							iAutoAuxStep3:=888;
							iNGSize:=iNGSize+1;		
						END_IF	
				END_IF
			END_IF
	ELSE
		BeltData[BeltNo.OverHang].iPanoramaNG:=0;
		BeltData[BeltNo.OverHang].fPoleNGSizeNo:=CCD_COM.Size.fPoleNGSizeNo; 
		stAlarm.arrLightWarn[5]:=TRUE;//尺寸CCD检测超时，请查看！
		iAutoAuxStep3:=888;
		iNGSize:=iNGSize+1;
	END_IF
888://
;
END_CASE


///////////////////////////////////////////////////////////冲R角定位检测//////////////////////////////////////////////////////////////////
CASE iAutoAuxStep4 OF
10://
	IF arrAxisCtrl[VirAxisNo.VirMain].Status.fActPos < fRecordMouldCCDInMainPos-fRecordMouldCCDInMainPosMod+360+ProductPar.parPublic.fMainPos-10 THEN//到下个周期250度以前有效			
		IF arrAxisCtrl[VirAxisNo.VirMain].Status.fActPos>=fRecordMouldCCDInMainPos+30 THEN		
			IF CCD_COM.Chamfer.iFinish=1 THEN
				CutMark_R[0]:=FALSE;
				TabData[TabNo.MouldPhoto].fTab_OffsetM:=CCD_COM.Chamfer.fTabXOffset;
				TabData[TabNo.MouldPhoto].fTab_OffsetY:=CCD_COM.Chamfer.fTabYOffset; //20240524SJ
				iAutoAuxStep4:=888;
			ELSIF CCD_COM.Chamfer.iFinish=2 THEN
				CutMark_R[0]:=FALSE;
				TabData[TabNo.MouldPhoto].fTab_OffsetM:=CCD_COM.Chamfer.fTabXOffset;//CCD抓不到极耳时，给NG，纠偏量给1个片宽
				TabData[TabNo.MouldPhoto].fTab_OffsetY:=CCD_COM.Chamfer.fTabYOffset; //20240524SJ
				TabData[TabNo.MouldPhoto].bTabOffsetNG_M:=TRUE;
				//stAlarm.arrLightWarn[1]:=TRUE;//冲R角CCD定位检测NG，请查看！
				iAutoAuxStep4:=888;	
			ELSIF CCD_COM.Chamfer.iFinish=3 THEN
				TabData[TabNo.MouldPhoto].bTabOffsetNG_M:=TRUE;
				CutMark_R[0]:=TRUE;
				iAutoAuxStep4:=888;	
			END_IF	
		END_IF		
	ELSE			
		//TabData[TabNo.MouldPhoto].fTab_OffsetM:=PolePar.fPoleWidth;
		TabData[TabNo.MouldPhoto].fTab_OffsetM:=0;//20240524SJ
		TabData[TabNo.MouldPhoto].bTabOffsetNG_M:=TRUE;
		stAlarm.arrLightWarn[2]:=TRUE;//冲R角CCD定位检测超时，请查看！		
		iAutoAuxStep4:=889;			
	END_IF
888:
	;
END_CASE

///////////////////////////////////////////////////////////裁切定位检测////////////////////////////////////////////////////////////////////
CASE iAutoAuxStep5 OF
10://
	IF arrAxisCtrl[VirAxisNo.VirMain].Status.fActPos < fRecordCuterCCDInMainPos-fRecordCuterCCDInMainPosMod+360+ProductPar.parPublic.fMainPos-10 THEN//到下个周期250度以前有效			
		IF arrAxisCtrl[VirAxisNo.VirMain].Status.fActPos>=fRecordCuterCCDInMainPos+30 THEN		
			IF CCD_COM.Cuter.iFinish=1 THEN	
				TabData[TabNo.CuterPhoto].fTab_OffsetC:=CCD_COM.Cuter.fTabXOffset;
				InteData[InteNo.Cuter-2].fTabIntervalC:=CCD_COM.Cuter.fTabWidth;
				iAutoAuxStep5:=100;
			ELSIF CCD_COM.Cuter.iFinish=2 THEN	
				TabData[TabNo.CuterPhoto].fTab_OffsetC:=CCD_COM.Cuter.fTabXOffset;
				InteData[InteNo.Cuter-2].fTabIntervalC:=CCD_COM.Cuter.fTabWidth;//CCD抓不到极耳时，给NG，左侧相机纠偏量给1个片宽,,片宽给0
				InteData[InteNo.Cuter-2].bIntervalFail_C:=TRUE;
				TabData[TabNo.CuterPhoto].bTabOffsetNG_C:=TRUE;
				//stAlarm.arrLightWarn[3]:=TRUE;//裁切CCD定位检测NG，请查看！		
				iAutoAuxStep5:=888;
			ELSIF CCD_COM.Cuter.iFinish=3 THEN	
	                 	TabData[TabNo.CuterPhoto].fTab_OffsetC:=CCD_COM.Cuter.fTabXOffset;
				InteData[InteNo.Cuter-2].fTabIntervalC:=CCD_COM.Cuter.fTabWidth;//CCD抓不到极耳时，给NG，左侧相机纠偏量给1个片宽,,片宽给0
				InteData[InteNo.Cuter-2].bIntervalFail_C:=TRUE;
				TabData[TabNo.CuterPhoto].bTabOffsetNG_C:=TRUE;
				//stAlarm.arrLightWarn[3]:=TRUE;//裁切CCD定位检测NG，请查看！		
				iAutoAuxStep5:=888;					
			END_IF	
		END_IF		
	ELSE			
		TabData[TabNo.CuterPhoto].fTab_OffsetC:=PolePar.fPoleWidth;
		InteData[InteNo.Cuter-2].fTabIntervalC:=0;	
		InteData[InteNo.Cuter-2].bIntervalFail_C:=TRUE;
		TabData[TabNo.CuterPhoto].bTabOffsetNG_C:=TRUE;
		PolePar.AddAlarm  :=PolePar.AddAlarm +1;
		stAlarm.arrLightWarn[4]:=TRUE;//裁切CCD定位检测超时，请查看！					
		iAutoAuxStep5:=889;		
	END_IF
	
100:

	IF CCD_COM.Cuter.iFinish=1 AND ( ABS(CCD_COM.Cuter.fTabWidth-PolePar.TabWidthBace)>=0.5 ) THEN
		Production.NGFlag[15]:=TRUE;
		iTabWidth_JS:=iTabWidth_JS+1;
		iAutoAuxStep5:=200;	
	ELSE
		iTabWidth_JS:=0;
		iAutoAuxStep5:=300;	
	END_IF
200:		
	IF iTabWidth_JS >=10 AND NOT ProductPar.iModeEN.bTabWidtNGoff THEN
		stAlarm.arrFlowAlarm[41]:=TRUE;//极片来料不良，请检查
		iTabWidth_JS:=0;
	END_IF
	Production.NGFlag[15]:=FALSE;
	iAutoAuxStep5:=888;	

300:
	iTabWidth_JS:=0;
	iAutoAuxStep5:=888;	
888:
	;	
	
	
END_CASE

////////////////////////////////////////////////////////////////线扫拍照触发////////////////////////////////////////////////////////////////
ttLinePhoto(CLK:=arrAxisCtrl[VirAxisNo.VirMain].Status.fModuloSetPos>=2  
						AND arrAxisCtrl[VirAxisNo.VirMain].Status.fModuloSetPos<=6 
						AND  arrAxisCtrl[VirAxisNo.VirMain].Status.Moving 
						AND  stDriverCam.bInSync         , Q=> );
IF ttLinePhoto.Q THEN
	CCD_COM.Scan.bSendMark:=FALSE;//PLC_To_PC上位机的发送数据标志
	IF NOT ProductPar.iModeEN.bCcdTcpEN AND NOT ProductPar.iModeEN.bLineScanCCDEN  THEN//线扫OK信号
		
		CCD_COM.Scan.iResult_IO_UP:=33;//复位线扫IO结果
		CCD_COM.Scan.iResult_IO_Down:=33;
		bLineScanResult1_UP:=FALSE;
		bLineScanResult2_UP:=FALSE;
		bLineScanResult1_Down:=FALSE;
		bLineScanResult2_Down:=FALSE;
		CCD_IO.boXSPhoto:=TRUE;//自动线扫启动
		CCD_Com.iLineScanPhotoCount:=CCD_Com.iLineScanPhotoCount+1;
		IF  NOT  ProductPar.iLineScanSel THEN
	    	iAutoAuxStep11:=10;
		END_IF
		fRecordLineineScanCCDInMainPos:=arrAxisCtrl[VirAxisNo.VirMain].Status.fActPos;																								
		fRecordLineineScanCCDInMainPosMod:=arrAxisCtrl[VirAxisNo.VirMain].Status.fModuloActPos;		
	END_IF	
END_IF	

rLineScan_UPTCP(CLK:=CCD_COM.Scan.iResult_UP<>33      , Q=> );
rLineScan_DownTCP(CLK:=CCD_COM.Scan.iResult_Down<>33 , Q=> );

IF ProductPar.iLineScanSel THEN
     IF rLineScan_UPTCP.Q THEN
		 IF CCD_COM.Scan.iResult_UP<>0 THEN
		    CCD_Com.iLineScanReceiveResultCount_UP:=CCD_Com.iLineScanReceiveResultCount_UP+1;
		 END_IF
	 END_IF

     IF rLineScan_DownTCP.Q THEN
		  IF CCD_COM.Scan.iResult_Down<>0 THEN
		     CCD_Com.iLineScanReceiveResultCount_Down:=CCD_Com.iLineScanReceiveResultCount_Down+1;
		  END_IF
	 END_IF

ELSE 
			IF  rLineScanOK_UP.Q  OR rLineScanNG_UP.Q THEN
				CCD_Com.iLineScanReceiveResultCount_UP:=CCD_Com.iLineScanReceiveResultCount_UP+1;
				fDA1:=        arrAxisCtrl[VirAxisNo.VirMain].Status.fModuloActPos;
			END_IF

		    IF  rLineScanOK_Down.Q  OR rLineScanNG_Down.Q THEN
				CCD_Com.iLineScanReceiveResultCount_Down:=CCD_Com.iLineScanReceiveResultCount_Down+1;
				fDA2:=        arrAxisCtrl[VirAxisNo.VirMain].Status.fModuloActPos;
			END_IF

END_IF			
			
	IF CCD_Com.bLineScanPhotoCountClear THEN
       CCD_Com.iLineScanPhotoCount:=0;
	   CCD_Com.iLineScanReceiveResultCount_UP:=0;
	   CCD_Com.iLineScanReceiveResultCount_Down:=0;
    END_IF		
			
				
CASE iAutoAuxStep11 OF
10://
	IF arrAxisCtrl[VirAxisNo.VirMain].Status.fModuloActPos>5 AND arrAxisCtrl[VirAxisNo.VirMain].Status.fModuloActPos < ProductPar.parPublic.fMainPos-15 THEN//到下个周期判断结果前有效
			IF rLineScanOK_UP.Q THEN
				bLineScanResult1_UP:=TRUE;
			END_IF
			IF rLineScanNG_UP.Q THEN
				bLineScanResult2_UP:=TRUE;
			END_IF

			IF rLineScanOK_Down.Q THEN
				bLineScanResult1_Down:=TRUE;
			END_IF
			IF rLineScanNG_Down.Q THEN
				bLineScanResult2_Down:=TRUE;
			END_IF	
	
		IF (bLineScanResult1_UP OR bLineScanResult2_UP) AND (bLineScanResult1_Down OR bLineScanResult2_Down) THEN
			iAutoAuxStep11:=888;
		END_IF
	
	ELSIF  arrAxisCtrl[VirAxisNo.VirMain].Status.fModuloActPos > 320 THEN
		IF NOT (bLineScanResult1_UP OR bLineScanResult2_UP) AND (bLineScanResult1_Down OR bLineScanResult2_Down) THEN  //AND NOT ProductPar.iModeEN.bCcdTcpEN AND NOT ProductPar.iModeEN.bLineScanCCDEN
			stAlarm.arrFlowAlarm[25]:=TRUE;//上线扫超时报警
		END_IF
		IF (bLineScanResult1_UP OR bLineScanResult2_UP) AND NOT (bLineScanResult1_Down OR bLineScanResult2_Down) THEN//	AND NOT ProductPar.iModeEN.bCcdTcpEN AND NOT ProductPar.iModeEN.bLineScanCCDEN 
			stAlarm.arrFlowAlarm[27]:=TRUE;//下线扫超时报警
		END_IF
		iAutoAuxStep11:=886;
	END_IF
	
END_CASE

///////////////////////////////////////////////////////////CCD标定流程////////////////////////////////////////////////////////////////////
IF stSysState.iMode=3 THEN
	CASE iAutoAuxStep10 OF 
	0://
		IF 	CCD_IO.bCalibrationsDo THEN
			bChaNoPhoto:=FALSE;
			bCutNoPhoto:=FALSE;			
			iAutoAuxStep10:=10;
		ELSIF NOT CCD_IO.bCalibrationsDo AND CCD_IO.bCalibrationsDo_Cha AND NOT CCD_IO.bCalibrationsDo_Cut THEN
			bChaNoPhoto:=FALSE;
			bCutNoPhoto:=TRUE;
			iAutoAuxStep10:=10;
		ELSIF NOT CCD_IO.bCalibrationsDo AND NOT CCD_IO.bCalibrationsDo_Cha AND CCD_IO.bCalibrationsDo_Cut THEN
			bChaNoPhoto:=TRUE;
			bCutNoPhoto:=FALSE;			
			iAutoAuxStep10:=10;
		END_IF
	10://
		CCD_IO.bDemRuning:=TRUE;
		CCD_COM.iDemCount:=1;//是否需要延时
		iAutoAuxStep10:=20;
	20://
		IF NOT bChaNoPhoto THEN
			CCD_COM.iDemResult_Cha:=0;
			CCD_IO.hmiChamferPhoto:=TRUE;
		END_IF
		IF NOT bCutNoPhoto THEN
			CCD_COM.iDemResult_Cut:=0;
			CCD_IO.hmiCuterPhoto:=TRUE;
		END_IF	
		iAutoAuxStep10:=30;
	30://
		IF tonAuto[17].Q THEN
			CCD_IO.hmiChamferPhoto:=FALSE;
			CCD_IO.hmiCuterPhoto:=FALSE;
			tonAuto[18].IN:=FALSE;
			iAutoAuxStep10:=40;
		END_IF
	40://
		IF (bChaNoPhoto  OR CCD_COM.iDemResult_Cha=1) AND (bCutNoPhoto OR CCD_COM.iDemResult_Cut=1) THEN
			tonAuto[18].IN:=FALSE;
			iAutoAuxStep10:=50;
		ELSIF (NOT bChaNoPhoto  AND CCD_COM.iDemResult_Cha=2) OR (NOT bCutNoPhoto AND CCD_COM.iDemResult_Cut=2) THEN
			tonAuto[18].IN:=FALSE;
			iAutoAuxStep10:=999;
		ELSE
			IF NOT tonAuto[18].Q THEN
				tonAuto[18].IN:=TRUE;
			ELSE
				tonAuto[18].IN:=FALSE;
				iAutoAuxStep10:=999;
			END_IF
		END_IF
	50://
		arrAxisCtrl[AxisNo.DriverDDR].Cmd.fPositon_of_Abs:=arrAxisCtrl[AxisNo.DriverDDR].Status.fActPos+FC_LengthToAngle(CCD_COM.fDemLength,PolePar.Machine.fMQDriverDiameter);
		arrAxisPar[AxisNo.DriverDDR].fVelocity_of_Abs:=5;
		arrAxisCtrl[AxisNo.DriverDDR].Cmd.bMoveAbs:=TRUE;
		iAutoAuxStep10:=60;
	60://
		IF arrAxisCtrl[AxisNo.DriverDDR].Status.Moving THEN
			CCD_COM.iDemCount:=2;
			iAutoAuxStep10:=70;
		END_IF
	70://
		IF NOT arrAxisCtrl[AxisNo.DriverDDR].Cmd.bMoveAbs AND arrAxisCtrl[AxisNo.DriverDDR].Status.NoMoving THEN
			iAutoAuxStep10:=80;
		END_IF
	80://
		IF NOT bChaNoPhoto THEN
			CCD_COM.iDemResult_Cha:=0;
			CCD_IO.hmiChamferPhoto:=TRUE;
		END_IF
		IF NOT bCutNoPhoto THEN
			CCD_COM.iDemResult_Cut:=0;
			CCD_IO.hmiCuterPhoto:=TRUE;
		END_IF	
		iAutoAuxStep10:=90;		
	90://
		IF tonAuto[17].Q THEN
			CCD_IO.hmiChamferPhoto:=FALSE;
			CCD_IO.hmiCuterPhoto:=FALSE;
			tonAuto[18].IN:=FALSE;
			iAutoAuxStep10:=100;
			arrAxisCtrl[AxisNo.DriverDDR].Cmd.fPositon_of_Abs:=arrAxisCtrl[AxisNo.DriverDDR].Status.fActPos-FC_LengthToAngle(CCD_COM.fDemLength,PolePar.Machine.fMQDriverDiameter);
			arrAxisPar[AxisNo.DriverDDR].fVelocity_of_Abs:=20;
			arrAxisCtrl[AxisNo.DriverDDR].Cmd.bMoveAbs:=TRUE;			
		END_IF	
	100://
		IF (bChaNoPhoto  OR CCD_COM.iDemResult_Cha=1) AND (bCutNoPhoto OR CCD_COM.iDemResult_Cut=1) THEN
			tonAuto[18].IN:=FALSE;
			iAutoAuxStep10:=666;
		ELSIF (NOT bChaNoPhoto  AND CCD_COM.iDemResult_Cha=2) OR (NOT bCutNoPhoto AND CCD_COM.iDemResult_Cut=2) THEN
			tonAuto[18].IN:=FALSE;
			iAutoAuxStep10:=999;
		ELSE
			IF NOT tonAuto[18].Q THEN
				tonAuto[18].IN:=TRUE;
			ELSE
				tonAuto[18].IN:=FALSE;
				iAutoAuxStep10:=999;
			END_IF
		END_IF	
	666://
		CCD_COM.iDemCount:=999;
		IF NOT bChaNoPhoto THEN
			CCD_IO.bCalibrationsDone_Cha:=TRUE;
		END_IF
		IF NOT bCutNoPhoto THEN
			CCD_IO.bCalibrationsDone_Cut:=TRUE;
		END_IF
		CCD_IO.bDemRuning:=FALSE;
		IF NOT arrAxisCtrl[AxisNo.DriverDDR].Cmd.bMoveAbs AND arrAxisCtrl[AxisNo.DriverDDR].Status.NoMoving THEN	
			iAutoAuxStep10:=0;
		END_IF
	999://
		CCD_COM.iDemCount:=999;
		IF NOT bChaNoPhoto THEN
			CCD_IO.bCalibrationsFals_Cha:=TRUE;
		END_IF
		IF NOT bCutNoPhoto THEN
			CCD_IO.bCalibrationsFals_Cut:=TRUE;
		END_IF
		CCD_IO.bDemRuning:=FALSE;	
		IF NOT arrAxisCtrl[AxisNo.DriverDDR].Cmd.bMoveAbs AND arrAxisCtrl[AxisNo.DriverDDR].Status.NoMoving THEN	
			iAutoAuxStep10:=0;
		END_IF
	END_CASE
ELSE
	CCD_COM.iDemCount:=999;
	CCD_IO.bDemRuning:=FALSE;
	iAutoAuxStep10:=0;		
END_IF


	(*
////////////////////////////////////////////////////////////////线扫拍照触发////////////////////////////////////////////////////////////////
ttLinePhoto(CLK:=arrAxisCtrl[VirAxisNo.VirMain].Status.fModuloSetPos>=2  
						AND arrAxisCtrl[VirAxisNo.VirMain].Status.fModuloSetPos<=6 
						AND  arrAxisCtrl[VirAxisNo.VirMain].Status.Moving 
						AND  stDriverCam.bInSync         , Q=> );
IF ttLinePhoto.Q THEN
	IF NOT ProductPar.iModeEN.bCcdTcpEN   THEN//线扫OK信号  //AND NOT ProductPar.iModeEN.bLineScanCCDEN
			IF BeltData[BeltNo.LineScanUp].iJumpCutNG=1 AND BeltData[BeltNo.LineScanUp+1].iJumpCutNG=1 AND BeltData[BeltNo.LineScanUp].fPoleNGSizeNo=30 THEN
				CCD_IO.hmiXSPhotoUp:=TRUE;//自动线扫启动
				CCD_COM.Scan.stPoleNoUp:=BeltData[BeltNo.LineScanUp].stPoleNo;			
			END_IF
			IF BeltData[BeltNo.LineScanDown].iJumpCutNG=1 AND BeltData[BeltNo.LineScanDown+1].iJumpCutNG=1 AND BeltData[BeltNo.LineScanDown].fPoleNGSizeNo=30 THEN
				CCD_IO.hmiXSPhotoDown:=TRUE;//自动线扫启动
				CCD_COM.Scan.stPoleNoDown:=BeltData[BeltNo.LineScanDown].stPoleNo;		
			END_IF		
			fRecordLineineScanCCDInMainPos:=arrAxisCtrl[VirAxisNo.VirMain].Status.fActPos;																								
			fRecordLineineScanCCDInMainPosMod:=arrAxisCtrl[VirAxisNo.VirMain].Status.fModuloActPos;	
	END_IF	
END_IF	
	*)


	
	
	
	
	(*


CASE iAutoAuxStep2 OF
100://
	IF NOT ProductPar.iModeEN.bEmptyRunEN THEN
		bMethodTenBufferEnable:=TRUE;
		iAutoAuxStep2:=200;
	ELSE
		bMethodTenBufferDisEnable:=TRUE;
		iAutoAuxStep2:=300;
	END_IF	
200://
	IF NOT bMethodTenBufferEnable THEN
		iAutoAuxStep2:=666;
	END_IF
300://
	IF NOT bMethodTenBufferDisEnable THEN
		iAutoAuxStep2:=350;
	END_IF
350://	
	arrCyCtrl[CYNo.DriverPressDDR].Cmd.bOFF:=TRUE;
	IF arrCyCtrl[CYNo.DriverPressDDR].Status.OFFState THEN
		iAutoAuxStep2:=666;
	END_IF
END_CASE
	
	*)
END_ACTION

ACTION F0512CarryAuto:
////////////////////////////////////////////////////////////////送片模式选择////////////////////////////////////////////////////////////////
IF ProductPar.iModeEN.bP2PartEN THEN
	iPoleCarryEver:=3;
ELSE
	iPoleCarryEver:=ProductPar.iModeEN.iCarryPoleMode;
END_IF
////////////////////////////////////////////////////////////////料况转化////////////////////////////////////////////////////////////////
bBelt_1[1]:=BeltData[BeltNo.SubBelt1].bHavePole;
bBelt_2[1]:=BeltData[BeltNo.SubBelt1-1].bHavePole;
bBelt_1[2]:=BeltData[BeltNo.SubBelt2].bHavePole;
bBelt_2[2]:=BeltData[BeltNo.SubBelt2-1].bHavePole;
bBelt_1[3]:=BeltData[BeltNo.SubBelt3].bHavePole;
bBelt_2[3]:=BeltData[BeltNo.SubBelt3-1].bHavePole;
////////////////////////////////////////////////////////////////送片皮带要料逻辑(皮带耦合,无料统计)    纯靠料况////////////////////////////////////////////////////////////////

bBelt_NO1:=bBelt_2[1] AND NOT bBelt_1[1] AND (   (bBelt_1[2] AND bBelt_1[3])  ) ;
bBelt_NO2:=bBelt_2[2] AND NOT bBelt_1[2] AND (  (bBelt_1[1] AND  bBelt_1[3])   ) ; 
bBelt_NO3:= ( bBelt_2[3] AND NOT bBelt_1[3] AND (   (bBelt_1[1] AND bBelt_1[2])  )  ) OR
			( bBelt_2[3] AND bBelt_1[3] AND (BeltData[BeltNo.SubBelt3].stPoleNo=''AND NOT ProductPar.iModeEN.bCcdTcpEN AND NOT ProductPar.iModeEN.bSizeCCDEN)
			AND (   (bBelt_1[1] AND bBelt_1[2]) ) ) ;


IF iPoleCarryEver=3 THEN
	bBelt3Need:=NOT BeltData[BeltNo.SubBelt3].bHavePole OR (BeltData[BeltNo.SubBelt3].bHavePole AND (BeltData[BeltNo.SubBelt3].stPoleNo=''AND NOT ProductPar.iModeEN.bCcdTcpEN AND NOT ProductPar.iModeEN.bSizeCCDEN) ) OR ProductPar.iModeEN.bP2PartEN;					
	bBelt2Need:=NOT BeltData[BeltNo.SubBelt2].bHavePole OR	 bBelt3Need;	
	
	IF bBelt_1[1] AND bBelt_1[2] AND (bBelt_1[3] AND (BeltData[BeltNo.SubBelt3].stPoleNo<>'' OR ProductPar.iModeEN.bCcdTcpEN OR ProductPar.iModeEN.bSizeCCDEN)) AND NOT ProductPar.iModeEN.bP2PartEN THEN
		iPoleNoHaveA:=0;
	ELSIF (bBelt_NO1 OR bBelt_NO2  OR bBelt_NO3 ) AND NOT ProductPar.iModeEN.bP2PartEN THEN
		iPoleNoHaveA:=1;
	ELSE
		iPoleNoHaveA:=2;	
	END_IF
ELSIF iPoleCarryEver=2 THEN
	bBelt3Need:=FALSE;
	bBelt2Need:=NOT BeltData[BeltNo.SubBelt2].bHavePole OR	 bBelt3Need;
	
	IF bBelt_1[1] AND bBelt_1[2]  AND NOT ProductPar.iModeEN.bP2PartEN   THEN
		iPoleNoHaveA:=0;
	ELSIF(
             (  bBelt_2[1] AND NOT bBelt_1[1] AND (  bBelt_1[2]  )   ) OR
			 (  bBelt_2[2] AND NOT bBelt_1[2] AND (  bBelt_1[1]  )   )
            )  AND NOT ProductPar.iModeEN.bP2PartEN  THEN
		iPoleNoHaveA:=1;
	ELSE
		iPoleNoHaveA:=2;	
	END_IF	
ELSE
	bBelt3Need:=FALSE;
	bBelt2Need:=FALSE OR	bBelt3Need;
	IF bBelt_1[1]  AND NOT ProductPar.iModeEN.bP2PartEN   THEN
		iPoleNoHaveA:=0;
	ELSIF ( bBelt_2[1] AND NOT bBelt_1[1] )  AND NOT ProductPar.iModeEN.bP2PartEN       THEN
		iPoleNoHaveA:=1;
	ELSE
		iPoleNoHaveA:=2;	
	END_IF							
END_IF

//取料位置有无片信号清理
IF rMQUse[11].Q THEN//叠台1
	BeltData[BeltNo.SubBelt1].bHavePole:=FALSE ;	
END_IF
IF rMQUse[12].Q THEN//叠台2
	BeltData[BeltNo.SubBelt2].bHavePole:=FALSE ;	
END_IF
IF rMQUse[13].Q THEN//叠台3
	BeltData[BeltNo.SubBelt3].bHavePole:=FALSE ;	
END_IF

(*****************减少取片等待时间*****************)
CASE iAutoAuxStep9 OF	
	100:
		tMQUse[1](IN:=FALSE , PT:=T#5S , Q=> , ET=> );
		IF iPartSelect=2 THEN
			iAutoAuxStep9:=200;//负极
		ELSE
			iAutoAuxStep9:=200;//300;//正极 20240509 CF
		END_IF
	200://负极不判断叠片主轴位置
		tMQUse[1](IN:=TRUE , PT:=T#5S , Q=> , ET=> );
		IF (InterPart.M1LockReady OR InterPart.M1JumpReady) AND (InterPart.M2LockReady OR InterPart.M2JumpReady) AND
			(InterPart.M3LockReady OR InterPart.M3JumpReady) THEN//OR tMQUse[1].Q 
			iAutoAuxStep9:=400;
		END_IF
	300://正极判断叠片主轴位置
		tMQUse[1](IN:=TRUE , PT:=T#5S , Q=> , ET=> );
		IF InterPart.M1LockReady AND InterPart.M2LockReady AND InterPart.M3LockReady THEN
			IF ABS(D_Sys.fM1MainSetPos-D_Sys.fM2MainSetPos)<1 AND ABS(D_Sys.fM1MainSetPos-D_Sys.fM3MainSetPos)<1
				AND ABS(D_Sys.fM2MainSetPos-D_Sys.fM3MainSetPos)<1 THEN
				iAutoAuxStep9:=400;//三个叠台同步
			END_IF
		ELSIF InterPart.M1LockReady AND InterPart.M2LockReady AND InterPart.M3JumpReady THEN
			IF ABS(D_Sys.fM1MainSetPos-D_Sys.fM2MainSetPos)<1 THEN
				iAutoAuxStep9:=400;// 1、2叠台同步
			END_IF
		ELSIF InterPart.M1LockReady AND InterPart.M2JumpReady AND InterPart.M3LockReady THEN
			IF ABS(D_Sys.fM1MainSetPos-D_Sys.fM3MainSetPos)<1 THEN
				iAutoAuxStep9:=400;//1、3叠台同步
			END_IF
		ELSIF InterPart.M1JumpReady AND InterPart.M2LockReady AND InterPart.M3LockReady THEN
			IF ABS(D_Sys.fM2MainSetPos-D_Sys.fM3MainSetPos)<1 THEN
				iAutoAuxStep9:=400;//2、3叠台同步
			END_IF
		ELSIF (InterPart.M1LockReady AND InterPart.M2JumpReady AND InterPart.M3JumpReady) 
				OR (InterPart.M1JumpReady AND InterPart.M2LockReady AND InterPart.M3JumpReady)
				OR (InterPart.M1JumpReady AND InterPart.M2JumpReady AND InterPart.M3LockReady) OR tMQUse[1].Q THEN
				iAutoAuxStep9:=400;//单个叠台
		END_IF
	400://允许取片信号   
		arrModPos[K10]:='';
		IF 	InterPart.M1LockReady AND (BeltData[BeltNo.SubBelt1].stPoleNo<>'' OR ProductPar.iModeEN.bCcdTcpEN OR ProductPar.iModeEN.bSizeCCDEN)  AND NOT bBelt1Taking THEN
			arrModPos[K10]:= CONCAT( arrModPos[K10], CONCAT( '     1#: ',REAL_TO_STRING(D_Sys.fM1MainSetPos)));	
			bMA10:=TRUE;
			iAutoAuxStep6:=10;
		END_IF
		IF 	InterPart.M2LockReady AND (BeltData[BeltNo.SubBelt2].stPoleNo<>''OR ProductPar.iModeEN.bCcdTcpEN OR ProductPar.iModeEN.bSizeCCDEN) AND NOT bBelt2Taking THEN
			arrModPos[K10]:= CONCAT( arrModPos[K10], CONCAT( '     2#: ',REAL_TO_STRING(D_Sys.fM2MainSetPos)));	
			bMA10:=TRUE;
			iAutoAuxStep7:=10;
		END_IF	
		IF 	InterPart.M3LockReady AND (BeltData[BeltNo.SubBelt3].stPoleNo<>''OR ProductPar.iModeEN.bCcdTcpEN OR ProductPar.iModeEN.bSizeCCDEN) AND NOT bBelt3Taking THEN
			arrModPos[K10]:= CONCAT( arrModPos[K10], CONCAT( '     3#: ',REAL_TO_STRING(D_Sys.fM3MainSetPos)));	
			bMA10:=TRUE;
			iAutoAuxStep8:=10;
		END_IF
		
		IF bMA10 THEN
			K10:=K10+1;
			IF K10>500 THEN
				K10:=1;
				MEMSET(ADR(arrModPos),0,SIZEOF(arrModPos));			
			END_IF
		   bMA10:=FALSE;
		END_IF
		
		iAutoAuxStep9:=666;	
END_CASE


///////////////////////////////////////////////////////////允许1叠台取料信号复位///////////////////////////////////////////////////////////////////20221101BYSJ
rtBelt1TakingReset1(CLK:=arrAxisCtrl[VirAxisNo.VirMain].Status.fModuloActPos>=10  AND   arrAxisCtrl[VirAxisNo.VirMain].Status.fModuloActPos<=20  AND 
                                      arrAxisCtrl[VirAxisNo.VirMain].Status.fSetVelo>=0.5          AND    bSubBelt1fratio      , Q=> );
rtBelt1TakingReset2(CLK:=arrAxisCtrl[VirAxisNo.VirMain].Status.fModuloActPos>=10  AND   arrAxisCtrl[VirAxisNo.VirMain].Status.fModuloActPos<=20  AND 
                                      arrAxisCtrl[VirAxisNo.VirMain].Status.fSetVelo>=0.5          AND    bSubBelt2fratio      , Q=> );									  
rtBelt1TakingReset3(CLK:=arrAxisCtrl[VirAxisNo.VirMain].Status.fModuloActPos>=10  AND   arrAxisCtrl[VirAxisNo.VirMain].Status.fModuloActPos<=20  AND 
                                      arrAxisCtrl[VirAxisNo.VirMain].Status.fSetVelo>=0.5          AND    bSubBelt3fratio      , Q=> );								  									  
IF  rtBelt1TakingReset1.Q THEN
	  InterPart.M1Allow:=FALSE;
      iAutoAuxStep6:=886;
END_IF	  
IF  rtBelt1TakingReset2.Q THEN
	  InterPart.M2Allow:=FALSE;
      iAutoAuxStep7:=886;
END_IF	  	  
IF  rtBelt1TakingReset3.Q THEN
	  InterPart.M3Allow:=FALSE;
      iAutoAuxStep8:=886;
END_IF	  



///////////////////////////////////////////////////////////允许1号叠台取料///////////////////////////////////////////////////////////////////
bBelt1Taking:=InterPart.M1Safety;
//DelayM1(IN:= , PT:=T#15MS , Q=> , ET=> );
IF rtAuto[7].Q THEN
	iAutoAuxStep6:=887;
	InterPart.M1Allow:=FALSE;
	//IF NOT InterPart.M1JumpReady THEN
		//BeltData[BeltNo.SubBelt1].bHavePole:=FALSE;
	//END_IF
END_IF

CASE iAutoAuxStep6 OF
10://
	IF NOT ProductPar.iModeEN.bP2PartEN AND NOT ProductPar.iModeEN.bEmptyRunEN  THEN
		InterPart.M1Allow:=TRUE;
	    iAutoAuxStep6:=20;
	ELSE
		 InterPart.M1Allow:=FALSE;
		  iAutoAuxStep6:=999;
	END_IF

20://   等待取片中信号
	IF bBelt1Taking THEN
		iAutoAuxStep6:=35;
	ELSIF (stSysState.iMode=3 OR NOT P2Interaction.P2M1Enable)AND NOT bBelt1Taking  THEN
		InterPart.M1Allow:=FALSE;
		iAutoAuxStep6:=888;
	END_IF
		
35: 
	IF     (  InterPart.M1Done OR  NOT  bBelt1Taking ) THEN//arrAxisCtrl[VirAxisNo.VirMain].Status.NoMoving AND
		InterPart.M1Allow:=FALSE;
		//IF NOT InterPart.M1JumpReady THEN
		//BeltData[BeltNo.SubBelt1].bHavePole:=FALSE ;
		//END_IF
		iAutoAuxStep6:=888;
	END_IF
END_CASE

(*
IF stSysState.iMode=3 AND bBelt1Taking  THEN
	InterPart.M1Allow:=FALSE;
	iAutoAuxStep6:=888;
END_IF
*)

BeltData[BeltNo.SubBelt1].bHavePole;
BeltData[BeltNo.SubBelt1-1].bHavePole;
BeltData[BeltNo.SubBelt1-2].bHavePole;



///////////////////////////////////////////////////////////允许2号叠台取料///////////////////////////////////////////////////////////////////

bBelt2Taking:=InterPart.M2Safety;
IF rtAuto[8].Q THEN
   	iAutoAuxStep7:=887;
	InterPart.M2Allow:=FALSE;
	//IF NOT InterPart.M2JumpReady THEN
 	//BeltData[BeltNo.SubBelt2].bHavePole:=FALSE;
	//END_IF
END_IF

CASE iAutoAuxStep7 OF
10://
	IF NOT ProductPar.iModeEN.bP2PartEN AND NOT ProductPar.iModeEN.bEmptyRunEN  THEN
		InterPart.M2Allow:=TRUE;
	    	iAutoAuxStep7:=20;
	ELSE
		 InterPart.M2Allow:=FALSE;
		  iAutoAuxStep7:=999;
	END_IF

20:////   等待取片中信号	
	IF bBelt2Taking THEN
		iAutoAuxStep7:=35;
	ELSIF (stSysState.iMode=3 OR NOT P2Interaction.P2M2Enable) AND NOT bBelt2Taking THEN
		InterPart.M2Allow:=FALSE;
		iAutoAuxStep7:=888;
	END_IF
	
35: 
	IF     (  InterPart.M2Done OR  NOT  bBelt2Taking ) THEN //arrAxisCtrl[VirAxisNo.VirMain].Status.NoMoving AND
		InterPart.M2Allow:=FALSE;
		//IF NOT InterPart.M2JumpReady THEN
		//BeltData[BeltNo.SubBelt2].bHavePole:=FALSE ;
		//END_IF
		iAutoAuxStep7:=888;
	END_IF
	 
END_CASE
(*
IF stSysState.iMode=3 AND bBelt2Taking AND InterPart.M2Safety THEN
	InterPart.M2Allow:=FALSE;
	iAutoAuxStep7:=888;
END_IF
*)


///////////////////////////////////////////////////////////允许3号叠台取料///////////////////////////////////////////////////////////////////
bBelt3Taking:=InterPart.M3Safety;
IF rtAuto[9].Q THEN
 	iAutoAuxStep8:=887;
	InterPart.M3Allow:=FALSE;
	//IF NOT InterPart.M3JumpReady THEN
	//BeltData[BeltNo.SubBelt3].bHavePole:=FALSE;
	//END_IF
END_IF


CASE iAutoAuxStep8 OF
10://
	IF NOT ProductPar.iModeEN.bP2PartEN AND NOT ProductPar.iModeEN.bEmptyRunEN  THEN
		InterPart.M3Allow:=TRUE;
	    iAutoAuxStep8:=20;
	ELSE
		 InterPart.M3Allow:=FALSE;
		  iAutoAuxStep8:=999;
	END_IF

20:////   等待取片中信号	
	IF bBelt3Taking THEN
		iAutoAuxStep8:=35;
	ELSIF (stSysState.iMode=3 OR NOT P2Interaction.P2M3Enable) AND NOT bBelt3Taking THEN
		InterPart.M3Allow:=FALSE;
		iAutoAuxStep8:=888;
	END_IF

35: 
	IF     (  InterPart.M3Done OR  NOT  bBelt3Taking ) THEN//arrAxisCtrl[VirAxisNo.VirMain].Status.NoMoving AND
		InterPart.M3Allow:=FALSE;
		//IF NOT InterPart.M3JumpReady THEN
		//BeltData[BeltNo.SubBelt3].bHavePole:=FALSE ;
		//END_IF
		iAutoAuxStep8:=888;
	END_IF
			
END_CASE
(*
IF stSysState.iMode=3 AND bBelt3Taking AND InterPart.M3Safety THEN
	InterPart.M3Allow:=FALSE;
	//bBelt3Taking:=FALSE;
	iAutoAuxStep8:=888;
END_IF
*)
END_ACTION

ACTION F0599AutoAux:
(*自动辅助*)
////////////////////////////////////微分&延时////////////////////////////////////
rtAuto[1](CLK:=SysPart.bAutoTen , Q=> );//自动触发
rtAuto[2](CLK:=stSysState.iMode=3 , Q=> );//手动
//rtAuto[3](CLK:=stSenser.biFlgBlue , Q=> );//蓝胶检测
//rtAuto[4](CLK:=CCD_COM.Scan.bLineScanNG , Q=> );//上线扫NG
//rtAuto[5](CLK:=CCD_COM.Scan.bLineScanNG , Q=> );//下线扫NG
rtAuto[6](CLK:=arrAxisCtrl[AxisNo.DriverDDR].Status.Moving , Q=> );//
rtAuto[7](CLK:=InterPart.M1Done , Q=> );//一号叠台取片完成
rtAuto[8](CLK:=InterPart.M2Done , Q=> );//二叠台取片完成
rtAuto[9](CLK:=InterPart.M3Done , Q=> );//三叠台取片完成



tonAuto[1](PT:=T#15S);//等待气缸动作/料盒顶升动作的时间
tonAuto[2](In:=stSenser.biSubBelt1Have,PT:=T#4MS);//皮带1倒数第二个工位有料延时
tonAuto[3](In:=NOT stSenser.biSubBelt1Have,PT:=T#4MS);//皮带1倒数第二个工位无料延时
tonAuto[4](In:=stSenser.biSubBelt2Have,PT:=T#4MS);//皮带2倒数第二个工位有料延时
tonAuto[5](In:=NOT stSenser.biSubBelt2Have,PT:=T#4MS);//皮带2倒数第二个工位无料延时
tonAuto[6](In:=stSenser.biSubBelt3Have,PT:=T#4MS);//皮带3倒数第二个工位有料延时
tonAuto[7](In:=NOT stSenser.biSubBelt3Have,PT:=T#4MS);//皮带3倒数第二个工位无料延时
tonAuto[8](In:=iAutoRunStep=2010,PT:=T#5MS);//主流程自动步序延时
//tonAuto[9](In:=arrCyCtrl[CYNo.NGBoxLock1].Cmd.bON OR arrCyCtrl[CYNo.NGBoxLock2].Cmd.bON,PT:=T#100MS);//NG归整气缸延时
tonAuto[10](In:=CCD_IO.boSizePhoto,PT:=T#50MS);//CCD拍照延时
tonAuto[11](In:=CCD_IO.boChamferPhoto,PT:=T#50MS);//CCD拍照延时
tonAuto[12](In:=CCD_IO.boCuterPhoto,PT:=T#50MS);//CCD拍照延时
//tonAuto[13](In:=iAutoAuxStep9=30,PT:=T#50MS);//NG料盒流程自动步序延时
//tonAuto[14](In:=iAutoAuxStep9=50,PT:=T#50MS);//NG料盒流程自动步序延时
//tonAuto[15](In:=stBtn.NGBoxStart AND SetpMotor.biBoxSensor ,PT:=T#500MS);//NG料盒满料后确认继续延时
//tonAuto[16](In:=NOT SetpMotor.biBoxSensor ,PT:=T#500MS);//NG料盒未到位延时
tonAuto[17](In:=iAutoAuxStep10=30 OR iAutoAuxStep10=90,PT:=T#50MS);//CCD标定流程步序延时
tonAuto[18](PT:=T#5S);//CCD标定流程延时
tonAuto[19](PT:=T#5S);//开机首次拍照延时
tonAuto[20](In:=CCD_IO.boXSPhoto,PT:=T#50MS);//皮带3倒数第二个工位无料延时
tonAuto[21](In:=iAutoRunStep=600,PT:=T#600MS);//皮带3倒数第二个工位无料延时
tonAuto[22](In:=,PT:=INT_TO_TIME(ProductPar.iModeEN.iNGcyCout)*60000);//单位时间内NG报警时间设定MIN
tonAuto[23](In:=stSenser.NGBoxFull,PT:=T#5S);//NG料盒满料报警
tonAuto[24](In:=bAnLaser,PT:=T#10S);
tonAuto[25](In:=bCaLaser,PT:=T#10S);
tonAuto[26](In:=bYellowPosTemp3,PT:=T#100MS);//黄标提示复位
tonAuto[27](In:=bYellowPosTemp4,PT:=T#100MS);//接带提示复位
tonAuto[28](In:=NOT YL_I[18],PT:=T#5S);//分段皮带3料盒满料报警
tonAuto[29](In:=NOT YL_I[19],PT:=T#5S);//分段皮带3料盒满料报警
tonAuto[30](In:=bYellowPosTemp6,PT:=T#100MS);//接带提示复位
tonAuto[31](In:=stSenser.NGboxsensor,PT:=T#2S);///NG踢废堵料报警
//上升沿
rMQUse[1](CLK:=stSenser.bYellowCheck_R1 , Q=> );//倒角前接带检测感应器	上	
rMQUse[2](CLK:=stSenser.bYellowCheck_R2  , Q=> );//倒角前接带检测感应器下
rMQUse[3](CLK:=stSenser.biFlgBlue, Q=> );//--R角前放卷蓝胶检测		
rMQUse[4](CLK:= arrAxisCtrl[VirAxisNo.VirMain].Status.Moving);//主轴启动上升沿
rMQUse[5](CLK:=iAutoRunStep=3000);//主程序步判断
rMQUse[6](CLK:=PolePar.bDemarcateBtn);//初始卷径标定触发上升沿
rMQUse[7](CLK:=arrCyCtrl[CyNo.Inflation_L].Io.DOStatus1);//左放卷气涨轴
rMQUse[8](CLK:=arrCyCtrl[CyNo.Inflation_R].Io.DOStatus1);//左放卷气涨轴
rMQUse[9](CLK:=stUwindTen.bError);//张力报警
rMQUse[10](CLK:=stSysState.iMode=1);//自动
rMQUse[11](CLK:=InterPart.M1PoleHave);//收到信号上升沿清叠台1取料位置有物料信号
rMQUse[12](CLK:=InterPart.M2PoleHave);//收到信号上升沿清叠台2取料位置有物料信号
rMQUse[13](CLK:=InterPart.M3PoleHave);//收到信号上升沿清叠台3取料位置有物料信号
rMQUse[14](CLK:=arrAxisCtrl[VirAxisNo.VirMain].Status.fModuloActPos>=150);////PLC_To_PC上位机的发送数据标志
rMQUse[15];
//下降沿
fMQUse[1](CLK:=stSenser.bYellowCheck_R1 , Q=> );//黄标检测---R角前
fMQUse[2](CLK:=stSenser.bYellowCheck_R2  , Q=> );//黄标检测---R角前
fMQUse[3](CLK:=stSenser.biFlgBlue, Q=> );//接带检测----R角前
fMQUse[4](CLK:= arrAxisCtrl[AxisNo.DriverDDR].Status.Moving);//DDR启动下降沿
fMQUse[5](CLK:= arrAxisCtrl[VirAxisNo.VirMain].Status.Moving);//主轴启动下降沿
fMQUse[7](CLK:=arrCyCtrl[CyNo.Inflation_L].Io.DOStatus1);//左放卷气涨轴
fMQUse[8](CLK:=arrCyCtrl[CyNo.Inflation_R].Io.DOStatus1);//左放卷气涨轴
 
IF stSysState.iMode=1 THEN
	Q107[11]:=FALSE;
	Q207[11]:=FALSE;
END_IF
//--CountClear
	IF iStopCount2>=30000 THEN
		iStopCount2 :=0;
	END_IF
	IF iOverCycleCount1>=30000 THEN
		iOverCycleCount1 :=0;
	END_IF
	IF iOverCycleCount2>=30000 THEN
		iOverCycleCount2 :=0;
	END_IF
	IF iOverCycleCount3>=30000 THEN
		iOverCycleCount3 :=0;
	END_IF
	IF iStopCount3>=30000 THEN
		iStopCount3 :=0;
	END_IF
	IF iStopCount>=30000 THEN
		iStopCount :=0;
	END_IF
	IF iPeaceAlarmCount1>=30000 THEN
		iPeaceAlarmCount1 :=0;
	END_IF
	IF iPeaceAlarmCount2>=30000 THEN
		iPeaceAlarmCount2 :=0;
	END_IF
	IF iPeaceAlarmCount3>=30000 THEN
		iPeaceAlarmCount3 :=0;
	END_IF
	
	
///主驱当前位置(转化为mm)
//fDriverDDRActPos:=FC_AngleToLength(arrAxisCtrl[AxisNo.DriverDDR].Status.fActPos,PolePar.Machine.fMQDriverDiameter);
fDriverDDRActPos:=(PI*PolePar.Machine.fMQDriverDiameter*arrAxisCtrl[AxisNo.DriverDDR].Status.fActPos)/360;

//PPM转化为M/min(转化)
PolePar.fMainHmiVel:=PolePar.iMainVel*PolePar.fPoleWidth/1000;
IF tonAuto[10].Q THEN
	CCD_IO.boSizePhoto:=FALSE;
END_IF
IF tonAuto[11].Q THEN
	CCD_IO.boChamferPhoto:=FALSE;
END_IF
IF tonAuto[12].Q THEN
	CCD_IO.boCuterPhoto:=FALSE;
END_IF
 IF tonAuto[20].Q THEN
	CCD_IO.boXSPhoto:=FALSE;
END_IF

////////////////////////////////////停止////////////////////////////////////
IF stSysState.Stoping AND SysPart.bAutoTen AND arrAxisCtrl[VirAxisNo.VirMain].Status.NoMoving AND 
	(iAutoRunStep>0 AND iAutoRunStep<600 OR iAutoRunStep>700 ) THEN
	iAutoRunStep:=600;
END_IF 

(*
//黄标检测,接带检测主驱位置记录
IF (rMQUse[1].Q OR rMQUse[2].Q )AND arrAxisCtrl[AxisNo.DriverDDR].Status.Moving THEN
	aYellowPos[1]:=fDriverDDRActPos;	
	FOR i4:=30 TO 2 BY -1 DO
		aYellowPos[i4]:=aYellowPos[i4-1];
	END_FOR	
END_IF
*)

//黄标检测,接带检测主驱位置记录
IF rMQUse[3].Q AND arrAxisCtrl[AxisNo.DriverDDR].Status.Moving AND NOT bYellowPosTemp1   THEN
    aYellowPosTemp1:=fDriverDDRActPos;
	aYellowPos[1]:=fDriverDDRActPos;	
	FOR i4:=30 TO 2 BY -1 DO
		aYellowPos[i4]:=aYellowPos[i4-1];
	END_FOR	
	bYellowPosTemp1:=TRUE;
	bYellowPosTemp3:=TRUE;
	Production.NGFlag[45]:=TRUE;//黄标计数
END_IF

IF ABS(fDriverDDRActPos-aYellowPosTemp1)>=12 THEN
	bYellowPosTemp1:=FALSE;
	Production.NGFlag[45]:=FALSE;//黄标计数
END_IF

IF tonAuto[26].Q THEN
	bYellowPosTemp3:=FALSE;
END_IF
(*
IF rMQUse[3].Q AND arrAxisCtrl[AxisNo.DriverDDR].Status.Moving THEN
	aTapePos[1]:=fDriverDDRActPos;	
	FOR i4:=30 TO 2 BY -1 DO
		aTapePos[i4]:=aTapePos[i4-1];
	END_FOR		
END_IF*)


//上	接带检测
IF rMQUse[1].Q AND arrAxisCtrl[AxisNo.DriverDDR].Status.Moving AND NOT bYellowPosTemp2 THEN
	aYellowPosTemp2:=fDriverDDRActPos;	
	aTapePos[1]:=fDriverDDRActPos;	
	FOR i4:=30 TO 2 BY -1 DO
		aTapePos[i4]:=aTapePos[i4-1];
	END_FOR		
	bYellowPosTemp2:=TRUE;
	bYellowPosTemp4:=TRUE;
	Production.NGFlag[43]:=TRUE;//接带计数
END_IF

IF ABS(fDriverDDRActPos-aYellowPosTemp2)>=20 THEN
	bYellowPosTemp2:=FALSE;
	Production.NGFlag[43]:=FALSE;//接带计数
END_IF

IF tonAuto[27].Q THEN
	bYellowPosTemp4:=FALSE;
END_IF

PolePar.fTape1_2:=555;
//下接带检测
IF rMQUse[2].Q  AND arrAxisCtrl[AxisNo.DriverDDR].Status.Moving AND NOT bYellowPosTemp5 THEN
	aYellowPosTemp2:=fDriverDDRActPos;	
	IF NOT bTapeMark THEN
		aTapepos2:=fDriverDDRActPos;
	END_IF
	aTapePos[1]:=fDriverDDRActPos+PolePar.fTape1_2;	
	FOR i4:=30 TO 2 BY -1 DO
		aTapePos[i4]:=aTapePos[i4-1];
	END_FOR		
	bYellowPosTemp5:=TRUE;
	bYellowPosTemp6:=TRUE;
	bTapeMark:=TRUE;
	Production.NGFlag[43]:=TRUE;//接带计数
END_IF

IF ABS(fDriverDDRActPos-aTapepos2)>=1900 THEN
	bTapeMark:=FALSE;
END_IF

IF ABS(fDriverDDRActPos-aYellowPosTemp2)>=20 THEN
	bYellowPosTemp5:=FALSE;
	Production.NGFlag[43]:=FALSE;//接带计数
END_IF

IF tonAuto[30].Q THEN
	bYellowPosTemp6:=FALSE;
END_IF


////////////////////////////////////////////////////////////////模具上模吹气///////////////////////////////////////////////////////////////
IF  stSysState.iMode=1 THEN
	IF arrAxisCtrl[AxisNo.Mould].Status.fModuloActPos>=arrAxisPar[AxisNo.Mould].arrTargetPoint[3] AND arrAxisCtrl[AxisNo.Mould].Status.fModuloActPos<arrAxisPar[AxisNo.Mould].arrTargetPoint[4]AND arrAxisCtrl[AxisNo.Mould].Status.Moving THEN
		arrCyCtrl[EVNo.MouldUpBlow].Cmd.bON:=TRUE;
		arrCyCtrl[EVNo.MouldUpBlow].Cmd.bOFF:=FALSE;
	ELSE
		arrCyCtrl[EVNo.MouldUpBlow].Cmd.bOFF:=TRUE;
		arrCyCtrl[EVNo.MouldUpBlow].Cmd.bON:=FALSE;
	END_IF
	////////////////////////////////////////////////////////////////模具下模吹气///////////////////////////////////////////////////////////////
	IF arrAxisCtrl[AxisNo.Mould].Status.fModuloActPos>=arrAxisPar[AxisNo.Mould].arrTargetPoint[5] AND arrAxisCtrl[AxisNo.Mould].Status.fModuloActPos<arrAxisPar[AxisNo.Mould].arrTargetPoint[6]AND arrAxisCtrl[AxisNo.Mould].Status.Moving THEN
		arrCyCtrl[EVNo.RJ_Blow].Cmd.bON:=TRUE;
		arrCyCtrl[EVNo.RJ_Blow].Cmd.bOFF:=FALSE;
	ELSE
		arrCyCtrl[EVNo.RJ_Blow].Cmd.bOFF:=TRUE;
		arrCyCtrl[EVNo.RJ_Blow].Cmd.bON:=FALSE;
	END_IF
END_IF

////////////////////////////////////////////////////////////////R角风刀吹气///////////////////////////////////////////////////////////////
IF 	stSysState.iMode=1 THEN
    IF  arrAxisCtrl[VirAxisNo.VirMain].Status.Moving THEN
		arrCyCtrl[EVNo.RJDustBlow  ].Cmd.bON:=TRUE;
		arrCyCtrl[EVNo.RJDustBlow  ].Cmd.bOFF:=FALSE;
	ELSE
		arrCyCtrl[EVNo.RJDustBlow  ].Cmd.bOFF:=TRUE;
		arrCyCtrl[EVNo.RJDustBlow  ].Cmd.bON:=FALSE;
	END_IF
END_IF
	
///////////////////////////分段送料皮带除尘毛刷////////////////////////////
IF arrAxisCtrl[AxisNo.	SubBelt1].Status.Moving AND fbSubBelt1Gear.fratio1>0 THEN
	arrDustMotor[MotorNo.FeduanbeltDust1].bRun_FW :=TRUE;
ELSE
	arrDustMotor[MotorNo.FeduanbeltDust1].bRun_FW :=FALSE;
END_IF

IF arrAxisCtrl[AxisNo.	SubBelt2].Status.Moving AND fbSubBelt2Gear.fratio1>0 THEN
	arrDustMotor[MotorNo.FeduanbeltDust2].bRun_FW :=TRUE;
ELSE
	arrDustMotor[MotorNo.FeduanbeltDust2].bRun_FW:=FALSE;
END_IF

IF arrAxisCtrl[AxisNo.	SubBelt3].Status.Moving AND fbSubBelt3Gear.fratio1>0 THEN
	arrDustMotor[MotorNo.FeduanbeltDust3].bRun_FW :=TRUE;
ELSE
	arrDustMotor[MotorNo.FeduanbeltDust3].bRun_FW :=FALSE;
END_IF

////////////////////////////////////急停////////////////////////////////////
IF stSysState.btnEstop AND arrAxisCtrl[VirAxisNo.VirMain].Status.Moving THEN
	arrAxisCtrl[AxisNo.CCDPressPush].Cmd. bHome:=FALSE;
	arrAxisCtrl[AxisNo.CCDPressPush].Cmd. bJog_Bw:=FALSE;	
	arrAxisCtrl[AxisNo.CCDPressPush].Cmd. bJog_Fw:=FALSE;		
	arrAxisCtrl[AxisNo.CCDPressPush].Cmd. bMoveAbs:=FALSE;		
	arrAxisCtrl[AxisNo.CCDPressPush].Cmd. bMoveRel:=FALSE;	
	arrAxisCtrl[AxisNo.CCDPressPush].Cmd. bMoveVelo:=FALSE;		
	arrAxisCtrl[AxisNo.CCDPressPush].Cmd.bMoveModulo:=FALSE;	
	arrAxisCtrl[AxisNo.CCDPressPush].Cmd. bSetPos:=FALSE;	 
	stCCDPressCam.bCamInExecute:=FALSE;   	
   	arrAxisCtrl[AxisNo.CCDPressPush].Cmd. iGoSetPos:=0;	  	
 	iHomestep:=0;
	iTensionStep:=0;
	iCamStep:=0;
	SysPart.Homeing:=FALSE;
	SysPart.Homed:=FALSE;	
	IF  arrAxisCtrl[AxisNo.CCDPressPush].Status.Moving  AND NOT arrAxisCtrl[AxisNo.CCDPressPush].Cmd.bStop   THEN//AND  NOT arrAxis[AxisNo.CCDPressPush] .Status.Coupled THEN   //对运动中的轴执行STOP
		arrAxisCtrl[AxisNo.CCDPressPush].Cmd. bStop:=TRUE;	
	END_IF;	
	arrAxisCtrl[AxisNo.Cuter].Cmd. bHome:=FALSE;
	arrAxisCtrl[AxisNo.Cuter].Cmd. bJog_Bw:=FALSE;	
	arrAxisCtrl[AxisNo.Cuter].Cmd. bJog_Fw:=FALSE;		
	arrAxisCtrl[AxisNo.Cuter].Cmd. bMoveAbs:=FALSE;		
	arrAxisCtrl[AxisNo.Cuter].Cmd. bMoveRel:=FALSE;	
	arrAxisCtrl[AxisNo.Cuter].Cmd. bMoveVelo:=FALSE;		
	arrAxisCtrl[AxisNo.Cuter].Cmd.bMoveModulo:=FALSE;	
	arrAxisCtrl[AxisNo.Cuter].Cmd. bSetPos:=FALSE;	    	
	arrAxisCtrl[AxisNo.Cuter].Cmd. iGoSetPos:=0;
	stCuterCam.bCamInExecute	:=FALSE;  		
	IF  arrAxisCtrl[AxisNo.Cuter].Status.Moving  AND NOT arrAxisCtrl[AxisNo.Cuter].Cmd.bStop   THEN//AND  NOT arrAxis[AxisNo.Cuter] .Status.Coupled THEN   //对运动中的轴执行STOP
	    	arrAxisCtrl[AxisNo.Cuter].Cmd. bStop:=TRUE;	
	END_IF;	
	arrAxisCtrl[AxisNo.Mould].Cmd. bHome:=FALSE;
	arrAxisCtrl[AxisNo.Mould].Cmd. bJog_Bw:=FALSE;	
	arrAxisCtrl[AxisNo.Mould].Cmd. bJog_Fw:=FALSE;		
	arrAxisCtrl[AxisNo.Mould].Cmd. bMoveAbs:=FALSE;		
	arrAxisCtrl[AxisNo.Mould].Cmd. bMoveRel:=FALSE;	
	arrAxisCtrl[AxisNo.Mould].Cmd. bMoveVelo:=FALSE;		
	arrAxisCtrl[AxisNo.Mould].Cmd.bMoveModulo:=FALSE;	
	arrAxisCtrl[AxisNo.Mould].Cmd. bSetPos:=FALSE;	    	
	arrAxisCtrl[AxisNo.Mould].Cmd. iGoSetPos:=0;	  
	stMouldCam.bCamInExecute:=FALSE;		
	IF  arrAxisCtrl[AxisNo.Mould].Status.Moving  AND NOT arrAxisCtrl[AxisNo.Mould].Cmd.bStop   THEN//AND  NOT arrAxis[AxisNo.Mould] .Status.Coupled THEN   //对运动中的轴执行STOP
	    	arrAxisCtrl[AxisNo.Mould].Cmd. bStop:=TRUE;	
	END_IF;		
	arrDustMotor[MotorNo.DDR_Dust].bRun_FW:=FALSE;																			
	arrDustMotor[MotorNo.CuterBeltDust].bRun_FW:=FALSE;																									
	arrDustMotor[MotorNo.NGReverseBeltDust].bRun_FW:=FALSE;																									
	arrDustMotor[MotorNo.DedustBeltDust].bRun_FW:=FALSE;																									
	arrDustMotor[MotorNo.DedustReverseBeltDust].bRun_FW:=FALSE;																									
	arrDustMotor[MotorNo.PoleBrushDust_U].bRun_FW:=FALSE;
	arrDustMotor[MotorNo.PoleBrushDust_D].bRun_FW:=FALSE;			
END_IF

//除尘启动  （包括皮带除尘电机）
IF NOT ProductPar.iModeEN.bDedustEN THEN
	IF arrAxisCtrl[VirAxisNo.VirMain].Status.Moving THEN		
		arrDustMotor[MotorNo.PoleBrushDust_U].bRun_FW:=TRUE;
		arrCyCtrl[EVNo.BrushDustVacuo_U].Cmd.bON:=TRUE;		
	
		arrCyCtrl[EVNo.WindDustBlow_U].Cmd.bON:=TRUE;
		arrCyCtrl[EVNo.WindDustVacuo_U].Cmd.bON:=TRUE;
	
		arrDustMotor[MotorNo.PoleBrushDust_D].bRun_FW:=TRUE;
		arrCyCtrl[EVNo.BrushDustVacuo_D].Cmd.bON:=TRUE;		
	
		arrCyCtrl[EVNo.WindDustBlow_D].Cmd.bON:=TRUE;
		arrCyCtrl[EVNo.WindDustVacuo_D].Cmd.bON:=TRUE;	
			
		arrDustMotor[MotorNo.DDR_Dust].bRun_FW:=TRUE;
		arrDustMotor[MotorNo.CuterBeltDust].bRun_FW:=TRUE;
		arrDustMotor[MotorNo.NGReverseBeltDust].bRun_FW:=TRUE;
		arrDustMotor[MotorNo.DedustBeltDust].bRun_FW:=TRUE;
		arrDustMotor[MotorNo.DedustReverseBeltDust].bRun_FW:=TRUE;				
	END_IF
	IF fMQUse[5].Q  THEN
		arrDustMotor[MotorNo.PoleBrushDust_U].bRun_FW:=FALSE;
		arrDustMotor[MotorNo.PoleBrushDust_D].bRun_FW:=FALSE;
		arrCyCtrl[EVNo.BrushDustVacuo_U].Cmd.bOff:=TRUE;		
		arrCyCtrl[EVNo.WindDustBlow_U].Cmd.bOff:=TRUE;
		arrCyCtrl[EVNo.WindDustVacuo_U].Cmd.bOff:=TRUE;		
		arrCyCtrl[EVNo.BrushDustVacuo_D].Cmd.bOff:=TRUE;	
		arrCyCtrl[EVNo.WindDustBlow_D].Cmd.bOff:=TRUE;
		arrCyCtrl[EVNo.WindDustVacuo_D].Cmd.bOff:=TRUE;
		
		arrDustMotor[MotorNo.DDR_Dust].bRun_FW:=FALSE;
		arrDustMotor[MotorNo.CuterBeltDust].bRun_FW:=FALSE;
		arrDustMotor[MotorNo.NGReverseBeltDust].bRun_FW:=FALSE;
		arrDustMotor[MotorNo.DedustBeltDust].bRun_FW:=FALSE;
		arrDustMotor[MotorNo.DedustReverseBeltDust].bRun_FW:=FALSE;			
	END_IF
ELSE
	IF  stSysState.iMode=1 THEN
		arrDustMotor[MotorNo.PoleBrushDust_U].bRun_FW:=FALSE;	
		arrDustMotor[MotorNo.PoleBrushDust_D].bRun_FW:=FALSE;		
		arrDustMotor[MotorNo.DDR_Dust].bRun_FW:=FALSE;
		arrDustMotor[MotorNo.CuterBeltDust].bRun_FW:=FALSE;
		arrDustMotor[MotorNo.NGReverseBeltDust].bRun_FW:=FALSE;
		arrDustMotor[MotorNo.DedustBeltDust].bRun_FW:=FALSE;
		arrDustMotor[MotorNo.DedustReverseBeltDust].bRun_FW:=FALSE;			
	END_IF
END_IF

//皮带运行前，气阀类状态
	IF rMQUse[5].Q THEN
		arrCyCtrl[EVNo.AreaArrayDustBlow].Cmd.bOFF:=TRUE;
		arrCyCtrl[EVNo.ConnectDustVacuo].Cmd.bOFF:=TRUE;
		arrCyCtrl[EVNo.LineSceneDustBlow].Cmd.bOFF:=TRUE;
		arrCyCtrl[EVNo.LineSceneDustVacuo].Cmd.bOFF:=TRUE;
		arrCyCtrl[EVNo.MouldDownAir].Cmd.bOFF:=TRUE;
		arrCyCtrl[EVNo.MouldDownVacuo].Cmd.bOFF:=TRUE;
	END_IF

	
//初始卷径手动标定程序
pRollWind:=SEL(PolePar.MQ.bWindSelect,ADR(arrAxis[AxisNo.UnWind_R]),ADR(arrAxis[AxisNo.UnWind_L]));
IF rMQUse[6].Q THEN
		DemarcateStep:=100;
	END_IF
CASE DemarcateStep OF

100://判断张力是否完成
	IF  stUwindTen.bTensionOK THEN
		DemarcateStep:=400;	
	ELSE
		DemarcateStep:=0;	
	END_IF
400:
	
	DemarcateStep:=450;
450://通过缓存电机移动距离与放卷轴放卷监督计算初始卷径---缓存到负极限位
	IF  arrAxisCtrl[AxisNo.BuffeLine].Cmd.arrbRealPoint[2] THEN
		arrAxisCtrl[AxisNo.BuffeLine].Cmd.iGoSetPos:=0;
		DemarcateStep:=500;	
	ELSE
		arrAxisCtrl[AxisNo.BuffeLine].Cmd.iGoSetPos:=2;		
	END_IF
500://判断摆杆是否到平衡位置
	IF  ABS (stAuxDriverTen.fDanserDegree -PolePar.MQ.AuxDriverTenBlancePos)<=5 THEN
		PolePar.rRollStartView:=pRollWind^.NcToPlc.ActPos;
		DemarcateStep:=600;
	END_IF
600://通过缓存电机移动距离与放卷轴放卷监督计算初始卷径---缓存到正极限位
	IF  arrAxisCtrl[AxisNo.BuffeLine].Cmd.arrbRealPoint[3] THEN
		arrAxisCtrl[AxisNo.BuffeLine].Cmd.iGoSetPos:=0;
		DemarcateStep:=700;	
	ELSE
		arrAxisCtrl[AxisNo.BuffeLine].Cmd.iGoSetPos:=3;		
	END_IF
700://判断摆杆是否到平衡位置
	IF  ABS (stAuxDriverTen.fDanserDegree -PolePar.MQ.AuxDriverTenBlancePos)<=5 THEN
		PolePar.rRollFinishView:=pRollWind^.NcToPlc.ActPos;
		DemarcateStep:=800;
	END_IF
800://计算
	PolePar.rRollView:=ABS(PolePar.rRollFinishView-PolePar.rRollStartView);//放卷运动总角度  
	PolePar.rRoll_L:=2*ABS(arrAxisPar[AxisNo.BuffeLine].arrTargetPoint[2]-arrAxisPar[AxisNo.BuffeLine].arrTargetPoint[3]);//缓存极片总长度(mm)	
	DemarcateStep:=900;
900:
	PolePar.rRollDia:=(360*PolePar.rRoll_L)/(Tc2_System.PI*PolePar.rRollView);
	DemarcateStep:=0;
END_CASE
(*	
	rRoll_L:REAL:=1000;//缓存极片总长度(mm)
	rRollStartView:REAL;//放卷开始角度
        rRollFinishView:REAL;//放卷结束角度 
	rRollView :REAL;//放卷运动总角度  
	rRollDia:REAL;//初始卷径(计数输出)
	bDemarcateBtn:BOOL;//标定开始按钮
*)	
	
CASE iAutoAuxStep1 OF
100://
	bMethodCamEnable:=TRUE;
	iAutoAuxStep1:=200;
200://
	IF NOT bMethodCamEnable THEN
		iAutoAuxStep1:=666;
	END_IF
END_CASE







(*****************************************************极耳基准20240101SJ*********************************************************************)
  rtTabSenser(CLK:=stSenser.bPoleCheck_R , Q=> );
  ftTabSenser(CLK:=stSenser.bPoleCheck_R , Q=> );
  (*
  IF  rtTabSenser.Q THEN
	  iCount100:=iCount100+1;
  END_IF
   IF  ftTabSenser.Q THEN
	  iCount101:=iCount101+1;
  END_IF 
  *)
 
  PolePar.fTabWidth:=53; //标准极耳宽度
  PolePar.fDriverStanderBasePos;//主驱动标准极耳下降沿位置
  PolePar.bDriverStanderBasePosEN;//自动找极耳基准屏蔽    1.等料带正常寻基准用    2. 屏蔽后不会 调整极耳

IF bTapeMark  THEN  
CASE  iTabOffsetStep  OF
	0: 
		  IF  arrAxisCtrl[VirAxisNo.VirMain].Status.fModuloSetPos>=2  AND   arrAxisCtrl[VirAxisNo.VirMain].Status.fModuloSetPos<=10  AND arrAxisCtrl[VirAxisNo.VirMain].Status.Moving AND  stDriverCam.bInSync   AND   
			   NOT ProductPar.iModeEN.bEmptyRunEN AND NOT ProductPar.iModeEN.bCcdTcpEN AND NOT ProductPar.iModeEN.bCuterOffsetEN AND stSysState.iMode=1     THEN
				 
			   bRecordPosM1:=FALSE;
			   bRecordPosM2:=FALSE;
			   fbReadTabCamSlavePos.Execute:=FALSE;
			   fVirMainSenserPos1:=0;
			   fVirMainSenserPos2:=0;  
			   IF K1>=50 THEN
				   K1:=1;
			   END_IF
	 
				IF  NOT   stSenser.bPoleCheck_R   THEN  
					 iTabOffsetStep:=100; // 启动前不在极耳上
				ELSE
					  iTabOffsetStep:=200; // 启动前就在极耳上
				END_IF
		   END_IF
	
	100:  //记录极耳上升沿，下降沿对应主轴位置
	   IF   arrAxisCtrl[VirAxisNo.VirMain].Status.fModuloSetPos<= ProductPar.parPublic.fMainPos  THEN
				IF  rtTabSenser.Q  AND NOT bRecordPosM1  THEN
					 fVirMainSenserPos1:=arrAxisCtrl[VirAxisNo.VirMain].Status.fModuloSetPos;
					 bRecordPosM1:=TRUE;
				END_IF
				IF  ftTabSenser.Q  AND NOT bRecordPosM2  THEN
					 fVirMainSenserPos2:=arrAxisCtrl[VirAxisNo.VirMain].Status.fModuloSetPos;
					 bRecordPosM2:=TRUE;
				END_IF    
			  IF  bRecordPosM1 AND  bRecordPosM2 THEN
				   iTabOffsetStep:=110;
			  END_IF
	   ELSIF  arrAxisCtrl[VirAxisNo.VirMain].Status.fModuloSetPos>ProductPar.parPublic.fMainPos-40  AND (NOT bRecordPosM1 OR NOT  bRecordPosM2) THEN //极耳检测异常 跳转到下个周期检测
			iTabOffsetStep:=0;
	   END_IF
	
	   
	  (********************以下程序大约需要10个扫描周期刷完***************************) 
	110://读取上升沿 主驱位置
	  IF  arrAxisCtrl[VirAxisNo.VirMain].Status.fModuloSetPos>=  ProductPar.parPublic.fMainPos-40  THEN   //避开Auto4   
	   fbReadTabCamSlavePos.MasterPosition:= fVirMainSenserPos1;
	   fbReadTabCamSlavePos.Execute:=TRUE;
	   iTabOffsetStep:=115;
	 END_IF  
	 115:
	  IF  fbReadTabCamSlavePos.Done THEN
		  fReadDriverPos1:= FC_AngleToLength(fbReadTabCamSlavePos.SlavePosition ,  PolePar.Machine.fMQDriverDiameter   )    ;
		  arrfReadDriverPos1[K1]:=fReadDriverPos1;
		  K1:=K1+1;
		  fbReadTabCamSlavePos.Execute:=FALSE;
		  iTabOffsetStep:=120;
	  ELSIF fbReadTabCamSlavePos.Error THEN //放弃此极耳检测
		  iTabOffsetStep:=0;
	  END_IF
	
	120://读取下降沿 主驱位置
	   fbReadTabCamSlavePos.MasterPosition:= fVirMainSenserPos2;
	   fbReadTabCamSlavePos.Execute:=TRUE;
	   iTabOffsetStep:=125;
	 125:
	  IF  fbReadTabCamSlavePos.Done THEN
		  fReadDriverPos2:=FC_AngleToLength( fbReadTabCamSlavePos.SlavePosition ,  PolePar.Machine.fMQDriverDiameter)  ;
		  arrfReadDriverPos2[K1]:=fReadDriverPos2;
		  fCalueTabWidth:=fReadDriverPos2-fReadDriverPos1;
		  iTabOffsetStep:=130;
	  ELSIF fbReadTabCamSlavePos.Error THEN //放弃此极耳检测
		  iTabOffsetStep:=0;
	  END_IF
	  
	  130: //判断极耳宽度是否在公差范围   如果在范围计算极耳下降沿主驱动位置与标准位置差值     
	   IF  fCalueTabWidth >=PolePar.fTabWidth-5 AND  fReadDriverPos2-fReadDriverPos1 <=PolePar.fTabWidth+5 THEN
			fTabOffset:= fReadDriverPos2- PolePar.fDriverStanderBasePos;      //如果>0 则 主驱补偿值>0才能让极耳恢复到标准值                      
		   iTabOffsetStep:=140;
	   ELSE  //极耳宽度异常
		   iTabOffsetStep:=0;
	  END_IF
	  
	  140:  //
		 IF  NOT   PolePar.bDriverStanderBasePosEN THEN
			 IF ABS(fTabOffset) >=30 THEN  //极耳严重偏离基准值
				  fDriverOffset:=            fTabOffset;  //给主驱补偿值用
				  bFlgTabPosOver:=TRUE;//  极耳严重偏移标志  给主驱补偿标志位用
				 // bFlgTabPosOver:=FALSE;//  极耳严重偏移标志  给主驱补偿标志位用
			ELSE
				  fDriverOffset:= 0;  //给主驱补偿值用
				  bFlgTabPosOver:=FALSE;//  极耳严重偏移标志  给主驱补偿标志位用	  
			 END_IF 	 
		ELSE
			 fDriverOffset:= 0;  //给主驱补偿值用
			 bFlgTabPosOver:=FALSE;//  极耳严重偏移标志
		 END_IF
		   iTabOffsetStep:=0;
			  
	200:	   
	   IF   arrAxisCtrl[VirAxisNo.VirMain].Status.fModuloSetPos<= ProductPar.parPublic.fMainPos  THEN
				IF  ftTabSenser.Q  AND NOT bRecordPosM2  THEN
					 fVirMainSenserPos2:=arrAxisCtrl[VirAxisNo.VirMain].Status.fModuloSetPos;
					 bRecordPosM2:=TRUE;
				END_IF    
			  IF    bRecordPosM2 THEN
				   iTabOffsetStep:=210;
			  END_IF
	   ELSIF  arrAxisCtrl[VirAxisNo.VirMain].Status.fModuloSetPos>ProductPar.parPublic.fMainPos-40   AND NOT  bRecordPosM2 THEN //极耳检测异常 跳转到下个周期检测
			iTabOffsetStep:=0;
	   END_IF  
		  
	  (********************以下程序大约需要10个扫描周期刷完***************************) 
	210://读取下降沿 主驱位置
	 IF  arrAxisCtrl[VirAxisNo.VirMain].Status.fModuloSetPos>=ProductPar.parPublic.fMainPos-40  THEN   //避开Auto4   
	   fbReadTabCamSlavePos.MasterPosition:= fVirMainSenserPos2;
	   fbReadTabCamSlavePos.Execute:=TRUE;
	   iTabOffsetStep:=225;
	   END_IF
	 225:
	  IF  fbReadTabCamSlavePos.Done THEN
		  fReadDriverPos2:=FC_AngleToLength( fbReadTabCamSlavePos.SlavePosition ,  PolePar.Machine.fMQDriverDiameter);
		  arrfReadDriverPos2[K1]:=fReadDriverPos2;
		 // fCalueTabWidth:=fReadDriverPos2-fReadDriverPos1;
		  iTabOffsetStep:=230;
	  ELSIF fbReadTabCamSlavePos.Error THEN //放弃此极耳检测
		  iTabOffsetStep:=0;
	  END_IF
	 
	 230: //判断极耳宽度是否在公差范围   如果在范围计算极耳下降沿主驱动位置与标准位置差值     
	  // IF  fCalueTabWidth >=fTabWidth-5 AND  fReadDriverPos2-fReadDriverPos1 <=fTabWidth+5 THEN
		   fTabOffset:= fReadDriverPos2- PolePar.fDriverStanderBasePos;      //如果>0 则 主驱补偿值>0才能让极耳恢复到标准值                      
		   iTabOffsetStep:=240;
	 //  ELSE  //极耳宽度异常
		  // iTabOffsetStep:=240;
	 // END_IF
	  
	  240:  // 
		 IF  NOT   PolePar.bDriverStanderBasePosEN THEN
			 IF ABS(fTabOffset) >=30 THEN  //极耳严重偏离基准值
				  fDriverOffset:=            fTabOffset;  //给主驱补偿值用
				  bFlgTabPosOver:=TRUE;//  极耳严重偏移标志  给主驱补偿标志位用
				 // bFlgTabPosOver:=FALSE;//  极耳严重偏移标志  给主驱补偿标志位用
			ELSE
				  fDriverOffset:= 0;  //给主驱补偿值用
				  bFlgTabPosOver:=FALSE;//  极耳严重偏移标志  给主驱补偿标志位用	  
			 END_IF 	 
		ELSE
			 fDriverOffset:= 0;  //给主驱补偿值用
			 bFlgTabPosOver:=FALSE;//  极耳严重偏移标志
		 END_IF
		   iTabOffsetStep:=0;  
			   
	END_CASE
ELSE
	bFlgTabPosOver:=FALSE;
END_IF

IF    PolePar.bDriverStanderBasePosEN THEN
	  bFlgTabPosOver:=FALSE;
END_IF


fbReadTabCamSlavePos.MasterPosition;
fbReadTabCamSlavePos(
	Execute:= , 
	CamTableID:=TableNo.Dirver , 
	MasterPosition:= , 
	Done=> , 
	Busy=> , 
	Error=> , 
	ErrorID=> , 
	SlavePosition=> , 
	SlaveVelocity=> , 
	SlaveAcceleration=> );

fbReadTabCamSlavePos.Done;
fbReadTabCamSlavePos.Error;
fbReadTabCamSlavePos.SlavePosition;


PolePar.fReadDriverPos3:=fReadDriverPos2;






(*****************************************************4连黄标尾料检测  SJ*********************************************************************)

ftTabSenser2(CLK:=stSenser.bFourYellowUP , Q=> );

IF ftTabSenser2.Q AND arrAxisCtrl[VirAxisNo.VirDriver].Status.Moving AND NOT bFourYellowFlg THEN
	arrfVirMainSenserPos[1]:=FC_AngleToLength(arrAxisCtrl[VirAxisNo.VirDriver].Status.fActPos , (PolePar.fPoleWidth+fbUwindTen.fCompensation)/Tc2_System.PI  )  ;
	bFourYellowFlg:=TRUE;
END_IF

arrfVirMainSenserPos[2]:=FC_AngleToLength(arrAxisCtrl[VirAxisNo.VirDriver].Status.fActPos , (PolePar.fPoleWidth+fbUwindTen.fCompensation)/Tc2_System.PI  )  ;
IF arrfVirMainSenserPos[2]-arrfVirMainSenserPos[1]>=10 THEN
	bFourYellowFlg:=FALSE;
END_IF

rtTabSenser2(CLK:=bFourYellowFlg , Q=> );
ProductPar.fYellowMackLength1; //相邻黄标后边距离
  
  //ProductPar.fDriverStanderBasePos;//主驱动标准极耳下降沿位置
  //ProductPar.bDriverStanderBasePosEN;//自动找极耳基准屏蔽    1.等料带正常寻基准用    2. 屏蔽后不会 调整极耳
  
CASE  iEndYellowMackStep  OF
	0: 
		IF  arrAxisCtrl[VirAxisNo.VirMain].Status.fModuloSetPos>=2  AND   arrAxisCtrl[VirAxisNo.VirMain].Status.fModuloSetPos<=10  AND arrAxisCtrl[VirAxisNo.VirMain].Status.Moving AND  stDriverCam.bInSync   THEN   
			iEndYellowMackStep:=100;
			nInt[2]	:=0;  
		END_IF
	
	100:  //记录极耳上升沿，下降沿对应主轴位置
		IF   arrAxisCtrl[VirAxisNo.VirMain].Status.fModuloSetPos<353   THEN
			
			IF  rtTabSenser2.Q THEN
				CASE nInt[2] OF
					0:
						arrbRecordPos[1] :=TRUE;
						nInt[2]	:=1;
					1:
						arrbRecordPos[2] :=TRUE;
						nInt[2]	:=2;
					2:
						arrbRecordPos[3] :=TRUE;
						nInt[2]	:=3;	
					3:
						arrbRecordPos[4] :=TRUE;
						nInt[2]	:=4;					
				END_CASE
			END_IF
		
		ELSIF 	  arrAxisCtrl[VirAxisNo.VirMain].Status.fModuloSetPos> 353 	 AND  arrAxisCtrl[VirAxisNo.VirMain].Status.fModuloSetPos< 360 THEN  
		
			IF arrbRecordPos[1]  AND arrbRecordPos[2] AND arrbRecordPos[3]  THEN  //至少有3个连续黄标
				stAlarm.arrFlowAlarm[42]:=bYellowMackAlarm:=TRUE;
				arrbRecordPos[1] :=arrbRecordPos[2] :=arrbRecordPos[3] :=arrbRecordPos[4]  := FALSE;
				iEndYellowMackStep:=0;
			ELSIF  arrbRecordPos[1]  AND arrbRecordPos[2] THEN    //当前周期检测出2个极耳 如果判定在设定间距则下个周期继续检
				nInt[2] :=2;
				iEndYellowMackStep:=200; //下个周期继续检测 极耳3
			ELSIF  arrbRecordPos[1]   THEN  // //当前周期检测出1个极耳  下个周期继续检黄标 2  3   4
				nInt[2] :=1;
				iEndYellowMackStep:=300; //下个周期继续检测 极耳2   3    4
			ELSE   //当前周期无黄标
				arrbRecordPos[1] :=arrbRecordPos[2] :=arrbRecordPos[3] :=arrbRecordPos[4]  := FALSE;
				iEndYellowMackStep:=0;
			END_IF
		
		END_IF
	
	
	200:    //下个周期继续检测极耳3  4
		IF  arrAxisCtrl[VirAxisNo.VirMain].Status.fModuloSetPos>=2  AND   arrAxisCtrl[VirAxisNo.VirMain].Status.fModuloSetPos<=10  AND arrAxisCtrl[VirAxisNo.VirMain].Status.Moving AND  stDriverCam.bInSync   THEN   
			iEndYellowMackStep:=210;   
		END_IF
		
	210:
		IF    arrAxisCtrl[VirAxisNo.VirMain].Status.fModuloSetPos< 180  THEN
			
			IF  rtTabSenser2.Q THEN
				CASE nInt[2] OF
					2:
						arrfVirMainSenserPos[3]:=     FC_AngleToLength(arrAxisCtrl[VirAxisNo.VirDriver].Status.fActPos ,     (PolePar.fPoleWidth+fbUwindTen.fCompensation)/Tc2_System.PI  )  ;
						arrbRecordPos[3] :=TRUE;
						nInt[2]	:=3;	
					3:
						arrfVirMainSenserPos[4]:=     FC_AngleToLength(arrAxisCtrl[VirAxisNo.VirDriver].Status.fActPos ,     (PolePar.fPoleWidth+fbUwindTen.fCompensation)/Tc2_System.PI  )  ;
						arrbRecordPos[4] :=TRUE;
						nInt[2]	:=4;					
				END_CASE
			END_IF
		
		ELSIF 	  arrAxisCtrl[VirAxisNo.VirMain].Status.fModuloSetPos> 180 	 AND  arrAxisCtrl[VirAxisNo.VirMain].Status.fModuloSetPos< 190 THEN 
  			 
			IF arrbRecordPos[1]  AND arrbRecordPos[2] AND arrbRecordPos[3]  THEN  //至少有3个连续黄标
				stAlarm.arrFlowAlarm[42]:=bYellowMackAlarm:=TRUE;
				arrbRecordPos[1] :=arrbRecordPos[2] :=arrbRecordPos[3] :=arrbRecordPos[4]  := FALSE;
				iEndYellowMackStep:=0;
			END_IF	
		
		ELSIF 	 arrAxisCtrl[VirAxisNo.VirMain].Status.fModuloSetPos> 190 	 AND  arrAxisCtrl[VirAxisNo.VirMain].Status.fModuloSetPos< 200   THEN   		
			arrbRecordPos[1] :=arrbRecordPos[2] :=arrbRecordPos[3] :=arrbRecordPos[4]  := FALSE;
			iEndYellowMackStep:=0;			
		END_IF
	
	300:  //下个周期继续检测 极耳2   3    4
		IF  arrAxisCtrl[VirAxisNo.VirMain].Status.fModuloSetPos>=2  AND   arrAxisCtrl[VirAxisNo.VirMain].Status.fModuloSetPos<=10  AND arrAxisCtrl[VirAxisNo.VirMain].Status.Moving AND  stDriverCam.bInSync   THEN   
			iEndYellowMackStep:=310;   
		END_IF
	
	310:
		IF   arrAxisCtrl[VirAxisNo.VirMain].Status.fModuloSetPos< 180   THEN
			
			IF  rtTabSenser2.Q THEN
				CASE nInt[2] OF
					1:
						arrbRecordPos[2] :=TRUE;
						nInt[2]	:=2;
					2:
						arrbRecordPos[3] :=TRUE;
						nInt[2]	:=3;	
					3:
						arrbRecordPos[4] :=TRUE;
						nInt[2]	:=4;					
				END_CASE
			END_IF	   
		
		ELSIF 	  arrAxisCtrl[VirAxisNo.VirMain].Status.fModuloSetPos> 180 	 AND  arrAxisCtrl[VirAxisNo.VirMain].Status.fModuloSetPos< 190 THEN  
		
			IF arrbRecordPos[1]  AND arrbRecordPos[2] AND arrbRecordPos[3]  THEN  //至少有3个连续黄
				stAlarm.arrFlowAlarm[42]:=bYellowMackAlarm:=TRUE;  
				arrbRecordPos[1] :=arrbRecordPos[2] :=arrbRecordPos[3] :=arrbRecordPos[4]  := FALSE;
				iEndYellowMackStep:=0;
			END_IF
			
		ELSIF 	  arrAxisCtrl[VirAxisNo.VirMain].Status.fModuloSetPos> 190 	 AND  arrAxisCtrl[VirAxisNo.VirMain].Status.fModuloSetPos< 200 THEN  			
			arrbRecordPos[1] :=arrbRecordPos[2] :=arrbRecordPos[3] :=arrbRecordPos[4]  := FALSE;
			iEndYellowMackStep:=0;	
		END_IF


END_CASE

(*
IF nInt[3]=1 THEN
	IF 160<arrAxisCtrl[VirAxisNo.VirMain].Status.fModuloSetPos AND arrAxisCtrl[VirAxisNo.VirMain].Status.fModuloSetPos<310 THEN
		arrCyCtrl[EvNo.	NGPushInsideAir	].Cmd.bON:=FALSE;//踢NG料打开
		arrCyCtrl[EvNo.	NGPushInsideAir	].Cmd.bOFF:=TRUE;//踢NG料关闭		
	ELSE
		arrCyCtrl[EvNo.	NGPushInsideAir	].Cmd.bON:=TRUE;//踢NG料打开
		arrCyCtrl[EvNo.	NGPushInsideAir	].Cmd.bOFF:=FALSE;//踢NG料关闭			
	END_IF
END_IF
BeltData[BeltNo.NGBox1+3].bHavePole;
BeltData[BeltNo.NGBox1+2].bHavePole;
*)


(*

(*****************************************************4连黄标尾料检测  SJ*********************************************************************)
  rtTabSenser2(CLK:=stSenser.bFourYellowUP , Q=> );
  ftTabSenser2(CLK:=stSenser.bFourYellowUP , Q=> );
  
  ProductPar.fYellowMackLength1; //相邻黄标后边距离
  
  //ProductPar.fDriverStanderBasePos;//主驱动标准极耳下降沿位置
  //ProductPar.bDriverStanderBasePosEN;//自动找极耳基准屏蔽    1.等料带正常寻基准用    2. 屏蔽后不会 调整极耳
  
CASE  iEndYellowMackStep  OF
0: 
      IF  arrAxisCtrl[VirAxisNo.VirMain].Status.fModuloSetPos>=2  AND   arrAxisCtrl[VirAxisNo.VirMain].Status.fModuloSetPos<=10  AND arrAxisCtrl[VirAxisNo.VirMain].Status.Moving AND  stDriverCam.bInSync   THEN   
            iEndYellowMackStep:=100;
			nInt[2]	:=0;  
       END_IF

100:  //记录极耳上升沿，下降沿对应主轴位置
  IF   arrAxisCtrl[VirAxisNo.VirMain].Status.fModuloSetPos< 353   THEN
	  IF  ftTabSenser2.Q THEN
	  		CASE nInt[2] OF
				0:
					arrfVirMainSenserPos[1]:=     FC_AngleToLength(arrAxisCtrl[VirAxisNo.VirDriver].Status.fActPos ,     (PolePar.fPoleWidth+fbUwindTen.fCompensation)/Tc2_System.PI  )  ;
					arrbRecordPos[1] :=TRUE;
					nInt[2]	:=1;
				1:
					arrfVirMainSenserPos[2]:=     FC_AngleToLength(arrAxisCtrl[VirAxisNo.VirDriver].Status.fActPos ,     (PolePar.fPoleWidth+fbUwindTen.fCompensation)/Tc2_System.PI  )  ;
					arrbRecordPos[2] :=TRUE;
					nInt[2]	:=2;
				2:
					arrfVirMainSenserPos[3]:=     FC_AngleToLength(arrAxisCtrl[VirAxisNo.VirDriver].Status.fActPos ,     (PolePar.fPoleWidth+fbUwindTen.fCompensation)/Tc2_System.PI  )  ;
					arrbRecordPos[3] :=TRUE;
					nInt[2]	:=3;	
				3:
					arrfVirMainSenserPos[4]:=     FC_AngleToLength(arrAxisCtrl[VirAxisNo.VirDriver].Status.fActPos ,     (PolePar.fPoleWidth+fbUwindTen.fCompensation)/Tc2_System.PI  )  ;
					arrbRecordPos[4] :=TRUE;
					nInt[2]	:=4;					
			END_CASE
		END_IF
		(*
			IF  ftTabSenser2.Q  AND NOT arrbRecordPos[1]  THEN
				 arrfVirMainSenserPos[1]:=     FC_AngleToLength(arrAxisCtrl[VirAxisNo.VirDriver].Status.fActPos ,     (PolePar.fPoleWidth+fbUwindTen.fCompensation)/Tc2_System.PI  )  ;
				 arrbRecordPos[1] :=TRUE;
			END_IF
			IF  ftTabSenser2.Q  AND  arrbRecordPos[1]  AND   NOT arrbRecordPos[2]  THEN
				 arrfVirMainSenserPos[2]:=     FC_AngleToLength(arrAxisCtrl[VirAxisNo.VirDriver].Status.fActPos ,     (PolePar.fPoleWidth+fbUwindTen.fCompensation)/Tc2_System.PI  )  ;
				 arrbRecordPos[2] :=TRUE;
			END_IF			
			IF  ftTabSenser2.Q  AND  arrbRecordPos[1]  AND  arrbRecordPos[2]     AND   NOT arrbRecordPos[3]  THEN
				 arrfVirMainSenserPos[3]:=     FC_AngleToLength(arrAxisCtrl[VirAxisNo.VirDriver].Status.fActPos ,     (PolePar.fPoleWidth+fbUwindTen.fCompensation)/Tc2_System.PI  )  ;
				 arrbRecordPos[3] :=TRUE;
			END_IF				
	    	IF  ftTabSenser2.Q  AND  arrbRecordPos[1]  AND  arrbRecordPos[2]    AND  arrbRecordPos[3]    AND   NOT arrbRecordPos[4]  THEN
				 arrfVirMainSenserPos[4]:=     FC_AngleToLength(arrAxisCtrl[VirAxisNo.VirDriver].Status.fActPos ,     (PolePar.fPoleWidth+fbUwindTen.fCompensation)/Tc2_System.PI  )  ;
				 arrbRecordPos[4] :=TRUE;
			 END_IF	
		*)					
ELSIF 	  arrAxisCtrl[VirAxisNo.VirMain].Status.fModuloSetPos> 353 	 AND  arrAxisCtrl[VirAxisNo.VirMain].Status.fModuloSetPos< 360 THEN  
			 
			IF arrbRecordPos[1]  AND arrbRecordPos[2] AND arrbRecordPos[3]  THEN  //至少有3个连续黄标
				      fD12:=arrfVirMainSenserPos[2] -arrfVirMainSenserPos[1];
			          fD23:=arrfVirMainSenserPos[3] -arrfVirMainSenserPos[2];
					  fD34:=arrfVirMainSenserPos[4] -arrfVirMainSenserPos[3];
					  
					 IF    ( arrfVirMainSenserPos[2] -arrfVirMainSenserPos[1] >=ProductPar.fYellowMackLength1-5  AND   arrfVirMainSenserPos[2] -arrfVirMainSenserPos[1] <=ProductPar.fYellowMackLength1+5 )  AND   
						   ( arrfVirMainSenserPos[3] -arrfVirMainSenserPos[2] >=ProductPar.fYellowMackLength1-5  AND   arrfVirMainSenserPos[3] -arrfVirMainSenserPos[2] <=ProductPar.fYellowMackLength1+5 )  THEN  //检测到3连黄标
						  bYellowMackAlarm:=TRUE;
						  
						   arrbRecordPos[1] :=arrbRecordPos[2] :=arrbRecordPos[3] :=arrbRecordPos[4]  := FALSE;
						  arrfVirMainSenserPos[1] :=arrfVirMainSenserPos[2] :=arrfVirMainSenserPos[3] :=arrfVirMainSenserPos[4]  := 0;  
							iEndYellowMackStep:=0;
				    ELSE    //不满足3连黄标条件   
						  arrbRecordPos[1] :=arrbRecordPos[2] :=arrbRecordPos[3] :=arrbRecordPos[4]  := FALSE;
						  arrfVirMainSenserPos[1] :=arrfVirMainSenserPos[2] :=arrfVirMainSenserPos[3] :=arrfVirMainSenserPos[4]  := 0;
						  iEndYellowMackStep:=0;
					 END_IF
			ELSIF  arrbRecordPos[1]  AND arrbRecordPos[2] THEN    //当前周期检测出2个极耳 如果判定在设定间距则下个周期继续检测
  		             fD12:=arrfVirMainSenserPos[2] -arrfVirMainSenserPos[1];
					 IF    ( arrfVirMainSenserPos[2] -arrfVirMainSenserPos[1] >=ProductPar.fYellowMackLength1-5  AND   arrfVirMainSenserPos[2] -arrfVirMainSenserPos[1] <=ProductPar.fYellowMackLength1+5 )  THEN   
					
							iEndYellowMackStep:=200; //下个周期继续检测 极耳3
				     ELSE    //不满足3连黄标条件   
						  arrbRecordPos[1] :=arrbRecordPos[2] :=arrbRecordPos[3] :=arrbRecordPos[4]  := FALSE;
						  arrfVirMainSenserPos[1] :=arrfVirMainSenserPos[2] :=arrfVirMainSenserPos[3] :=arrfVirMainSenserPos[4]  := 0;
						  iEndYellowMackStep:=0;
					 END_IF
					 
			ELSIF  arrbRecordPos[1]   THEN  // //当前周期检测出1个极耳  下个周期继续检黄标 2  3   4
		              iEndYellowMackStep:=300; //下个周期继续检测 极耳2   3    4
	
			ELSE   //当前周期无黄标
					 arrbRecordPos[1] :=arrbRecordPos[2] :=arrbRecordPos[3] :=arrbRecordPos[4]  := FALSE;
					arrfVirMainSenserPos[1] :=arrfVirMainSenserPos[2] :=arrfVirMainSenserPos[3] :=arrfVirMainSenserPos[4]  := 0;
			         iEndYellowMackStep:=0;
			
			END_IF

   END_IF

  
200:    //下个周期继续检测极耳3  4
      IF  arrAxisCtrl[VirAxisNo.VirMain].Status.fModuloSetPos>=2  AND   arrAxisCtrl[VirAxisNo.VirMain].Status.fModuloSetPos<=10  AND arrAxisCtrl[VirAxisNo.VirMain].Status.Moving AND  stDriverCam.bInSync   THEN   
            iEndYellowMackStep:=210;   
       END_IF
210:
IF    arrAxisCtrl[VirAxisNo.VirMain].Status.fModuloSetPos< 180  THEN
	IF  ftTabSenser2.Q THEN
			CASE nInt[2] OF
				0:
					arrfVirMainSenserPos[1]:=     FC_AngleToLength(arrAxisCtrl[VirAxisNo.VirDriver].Status.fActPos ,     (PolePar.fPoleWidth+fbUwindTen.fCompensation)/Tc2_System.PI  )  ;
					arrbRecordPos[1] :=TRUE;
					nInt[2]	:=1;
				1:
					arrfVirMainSenserPos[2]:=     FC_AngleToLength(arrAxisCtrl[VirAxisNo.VirDriver].Status.fActPos ,     (PolePar.fPoleWidth+fbUwindTen.fCompensation)/Tc2_System.PI  )  ;
					arrbRecordPos[2] :=TRUE;
					nInt[2]	:=2;
				2:
					arrfVirMainSenserPos[3]:=     FC_AngleToLength(arrAxisCtrl[VirAxisNo.VirDriver].Status.fActPos ,     (PolePar.fPoleWidth+fbUwindTen.fCompensation)/Tc2_System.PI  )  ;
					arrbRecordPos[3] :=TRUE;
					nInt[2]	:=3;	
				3:
					arrfVirMainSenserPos[4]:=     FC_AngleToLength(arrAxisCtrl[VirAxisNo.VirDriver].Status.fActPos ,     (PolePar.fPoleWidth+fbUwindTen.fCompensation)/Tc2_System.PI  )  ;
					arrbRecordPos[4] :=TRUE;
					nInt[2]	:=4;					
			END_CASE
	END_IF
			(*
			IF  ftTabSenser2.Q  AND  arrbRecordPos[1]  AND  arrbRecordPos[2]     AND   NOT arrbRecordPos[3]  THEN
				 arrfVirMainSenserPos[3]:=     FC_AngleToLength(arrAxisCtrl[VirAxisNo.VirDriver].Status.fActPos ,     (PolePar.fPoleWidth+fbUwindTen.fCompensation)/Tc2_System.PI  )  ;
				 arrbRecordPos[3] :=TRUE;
			END_IF				
	    	IF  ftTabSenser2.Q  AND  arrbRecordPos[1]  AND  arrbRecordPos[2]    AND  arrbRecordPos[3]    AND   NOT arrbRecordPos[4]  THEN
				 arrfVirMainSenserPos[4]:=     FC_AngleToLength(arrAxisCtrl[VirAxisNo.VirDriver].Status.fActPos ,     (PolePar.fPoleWidth+fbUwindTen.fCompensation)/Tc2_System.PI  )  ;
				 arrbRecordPos[4] :=TRUE;
			 END_IF
		*)									 
ELSIF 	  arrAxisCtrl[VirAxisNo.VirMain].Status.fModuloSetPos> 180 	 AND  arrAxisCtrl[VirAxisNo.VirMain].Status.fModuloSetPos< 190 THEN   			 
			 	IF arrbRecordPos[1]  AND arrbRecordPos[2] AND arrbRecordPos[3]  THEN  //至少有3个连续黄标
				      fD12:=arrfVirMainSenserPos[2] -arrfVirMainSenserPos[1];
			          fD12:=arrfVirMainSenserPos[3] -arrfVirMainSenserPos[2];
					  fD12:=arrfVirMainSenserPos[4] -arrfVirMainSenserPos[3];
					  
					 IF    ( arrfVirMainSenserPos[2] -arrfVirMainSenserPos[1] >=ProductPar.fYellowMackLength1-5  AND   arrfVirMainSenserPos[2] -arrfVirMainSenserPos[1] <=ProductPar.fYellowMackLength1+5 )  AND   
						   ( arrfVirMainSenserPos[3] -arrfVirMainSenserPos[2] >=ProductPar.fYellowMackLength1-5  AND   arrfVirMainSenserPos[3] -arrfVirMainSenserPos[2] <=ProductPar.fYellowMackLength1+5 )  THEN  //检测到3连黄标
						  bYellowMackAlarm:=TRUE;
						   arrbRecordPos[1] :=arrbRecordPos[2] :=arrbRecordPos[3] :=arrbRecordPos[4]  := FALSE;
						  arrfVirMainSenserPos[1] :=arrfVirMainSenserPos[2] :=arrfVirMainSenserPos[3] :=arrfVirMainSenserPos[4]  := 0;  
							iEndYellowMackStep:=0;
				    ELSE    //不满足3连黄标条件   
						  arrbRecordPos[1] :=arrbRecordPos[2] :=arrbRecordPos[3] :=arrbRecordPos[4]  := FALSE;
						  arrfVirMainSenserPos[1] :=arrfVirMainSenserPos[2] :=arrfVirMainSenserPos[3] :=arrfVirMainSenserPos[4]  := 0;
						  iEndYellowMackStep:=100;
					 END_IF			 	 
			    END_IF	
				
ELSIF 	 arrAxisCtrl[VirAxisNo.VirMain].Status.fModuloSetPos> 190 	 AND  arrAxisCtrl[VirAxisNo.VirMain].Status.fModuloSetPos< 200   THEN   		
						  arrbRecordPos[1] :=arrbRecordPos[2] :=arrbRecordPos[3] :=arrbRecordPos[4]  := FALSE;
						  arrfVirMainSenserPos[1] :=arrfVirMainSenserPos[2] :=arrfVirMainSenserPos[3] :=arrfVirMainSenserPos[4]  := 0;
						  iEndYellowMackStep:=100;			
 END_IF
   
 
 
 
 
 300:  //下个周期继续检测 极耳2   3    4
       IF  arrAxisCtrl[VirAxisNo.VirMain].Status.fModuloSetPos>=2  AND   arrAxisCtrl[VirAxisNo.VirMain].Status.fModuloSetPos<=10  AND arrAxisCtrl[VirAxisNo.VirMain].Status.Moving AND  stDriverCam.bInSync   THEN   
            iEndYellowMackStep:=310;   
       END_IF

 310:
   IF   arrAxisCtrl[VirAxisNo.VirMain].Status.fModuloSetPos< 180   THEN
		IF  ftTabSenser2.Q THEN
				CASE nInt[2] OF
					0:
						arrfVirMainSenserPos[1]:=     FC_AngleToLength(arrAxisCtrl[VirAxisNo.VirDriver].Status.fActPos ,     (PolePar.fPoleWidth+fbUwindTen.fCompensation)/Tc2_System.PI  )  ;
						arrbRecordPos[1] :=TRUE;
						nInt[2]	:=1;
					1:
						arrfVirMainSenserPos[2]:=     FC_AngleToLength(arrAxisCtrl[VirAxisNo.VirDriver].Status.fActPos ,     (PolePar.fPoleWidth+fbUwindTen.fCompensation)/Tc2_System.PI  )  ;
						arrbRecordPos[2] :=TRUE;
						nInt[2]	:=2;
					2:
						arrfVirMainSenserPos[3]:=     FC_AngleToLength(arrAxisCtrl[VirAxisNo.VirDriver].Status.fActPos ,     (PolePar.fPoleWidth+fbUwindTen.fCompensation)/Tc2_System.PI  )  ;
						arrbRecordPos[3] :=TRUE;
						nInt[2]	:=3;	
					3:
						arrfVirMainSenserPos[4]:=     FC_AngleToLength(arrAxisCtrl[VirAxisNo.VirDriver].Status.fActPos ,     (PolePar.fPoleWidth+fbUwindTen.fCompensation)/Tc2_System.PI  )  ;
						arrbRecordPos[4] :=TRUE;
						nInt[2]	:=4;					
				END_CASE
		END_IF	   
(*	   
			IF  ftTabSenser2.Q  AND  arrbRecordPos[1]  AND   NOT arrbRecordPos[2]  THEN
				 arrfVirMainSenserPos[2]:=     FC_AngleToLength(arrAxisCtrl[VirAxisNo.VirDriver].Status.fActPos ,     (PolePar.fPoleWidth+fbUwindTen.fCompensation)/Tc2_System.PI  )  ;
				 arrbRecordPos[2] :=TRUE;
			END_IF			
			IF  ftTabSenser2.Q  AND  arrbRecordPos[1]  AND  arrbRecordPos[2]     AND   NOT arrbRecordPos[3]  THEN
				 arrfVirMainSenserPos[3]:=     FC_AngleToLength(arrAxisCtrl[VirAxisNo.VirDriver].Status.fActPos ,     (PolePar.fPoleWidth+fbUwindTen.fCompensation)/Tc2_System.PI  )  ;
				 arrbRecordPos[3] :=TRUE;
			END_IF				
	    	IF  ftTabSenser2.Q  AND  arrbRecordPos[1]  AND  arrbRecordPos[2]    AND  arrbRecordPos[3]    AND   NOT arrbRecordPos[4]  THEN
				 arrfVirMainSenserPos[4]:=     FC_AngleToLength(arrAxisCtrl[VirAxisNo.VirDriver].Status.fActPos ,     (PolePar.fPoleWidth+fbUwindTen.fCompensation)/Tc2_System.PI  )  ;
				 arrbRecordPos[4] :=TRUE;
			 END_IF
*)						
ELSIF 	  arrAxisCtrl[VirAxisNo.VirMain].Status.fModuloSetPos> 180 	 AND  arrAxisCtrl[VirAxisNo.VirMain].Status.fModuloSetPos< 190 THEN  
			 
			IF arrbRecordPos[1]  AND arrbRecordPos[2] AND arrbRecordPos[3]  THEN  //至少有3个连续黄标
				      fD12:=arrfVirMainSenserPos[2] -arrfVirMainSenserPos[1];
			          fD12:=arrfVirMainSenserPos[3] -arrfVirMainSenserPos[2];
					  fD12:=arrfVirMainSenserPos[4] -arrfVirMainSenserPos[3];	  
					 IF    ( arrfVirMainSenserPos[2] -arrfVirMainSenserPos[1] >=ProductPar.fYellowMackLength1-5  AND   arrfVirMainSenserPos[2] -arrfVirMainSenserPos[1] <=ProductPar.fYellowMackLength1+5 )  AND   
						   ( arrfVirMainSenserPos[3] -arrfVirMainSenserPos[2] >=ProductPar.fYellowMackLength1-5  AND   arrfVirMainSenserPos[3] -arrfVirMainSenserPos[2] <=ProductPar.fYellowMackLength1+5 )  THEN  //检测到3连黄标
						  bYellowMackAlarm:=TRUE;  
						   arrbRecordPos[1] :=arrbRecordPos[2] :=arrbRecordPos[3] :=arrbRecordPos[4]  := FALSE;
						  arrfVirMainSenserPos[1] :=arrfVirMainSenserPos[2] :=arrfVirMainSenserPos[3] :=arrfVirMainSenserPos[4]  := 0;  
							iEndYellowMackStep:=0;
				    ELSE    //不满足3连黄标条件   
						  arrbRecordPos[1] :=arrbRecordPos[2] :=arrbRecordPos[3] :=arrbRecordPos[4]  := FALSE;
						  arrfVirMainSenserPos[1] :=arrfVirMainSenserPos[2] :=arrfVirMainSenserPos[3] :=arrfVirMainSenserPos[4]  := 0;
						  iEndYellowMackStep:=100;
					 END_IF
		  ELSE   //当前周期无黄标
					 arrbRecordPos[1] :=arrbRecordPos[2] :=arrbRecordPos[3] :=arrbRecordPos[4]  := FALSE;
					arrfVirMainSenserPos[1] :=arrfVirMainSenserPos[2] :=arrfVirMainSenserPos[3] :=arrfVirMainSenserPos[4]  := 0;
			         iEndYellowMackStep:=100;
			END_IF

ELSIF 	  arrAxisCtrl[VirAxisNo.VirMain].Status.fModuloSetPos> 190 	 AND  arrAxisCtrl[VirAxisNo.VirMain].Status.fModuloSetPos< 200 THEN  			
			arrbRecordPos[1] :=arrbRecordPos[2] :=arrbRecordPos[3] :=arrbRecordPos[4]  := FALSE;
			arrfVirMainSenserPos[1] :=arrfVirMainSenserPos[2] :=arrfVirMainSenserPos[3] :=arrfVirMainSenserPos[4]  := 0;
		    iEndYellowMackStep:=100;	
 END_IF

   
END_CASE

*)
END_ACTION

ACTION F05Rectifydev:

(******************************************************************极片纠偏V2  SJ*****************************************************************************)
//极片纠偏条件
fbRectifyGM.bRecEn:=   (  (   (arrAxisCtrl[VirAxisNo.VirMain].Status.fModuloSetPos>=5  AND arrAxisCtrl[VirAxisNo.VirMain].Status.fModuloSetPos<80) OR 
                                               (arrAxisCtrl[VirAxisNo.VirMain].Status.fModuloSetPos>=180  AND arrAxisCtrl[VirAxisNo.VirMain].Status.fModuloSetPos<250)  )      AND
	                                          arrAxisCtrl[VirAxisNo.VirMain].Status.Moving AND  stDriverCam.bInSync AND NOT ProductPar.iModeEN.bMouldYRecEN AND
                                              NOT bCyDDRMark AND NOT  RecYRules[1] )       ;
											  
(*fbRectifyGM.bRecEn:=   (  (   (arrAxisCtrl[VirAxisNo.VirMain].Status.fModuloSetPos>=5  AND arrAxisCtrl[VirAxisNo.VirMain].Status.fModuloSetPos<80) OR 
                                               (arrAxisCtrl[VirAxisNo.VirMain].Status.fModuloSetPos>=180  AND arrAxisCtrl[VirAxisNo.VirMain].Status.fModuloSetPos<250)  )      AND
	                                          arrAxisCtrl[VirAxisNo.VirMain].Status.Moving AND  stDriverCam.bInSync AND NOT ProductPar.iModeEN.bMouldYRecEN  AND NOT  RecYRules[1] )       ;*)											  
								  
//黄标不纠偏范围判断,,,-170指黄标感应器高裁切距离-170=黄标感应器到纠偏传感器的距离,,,即纠偏传感器到裁切切刀距离为170
	FOR i9:=1 TO 20  DO	
		(*
		IF (PolePar.fPoleWidth-50<=(aYellowPos[i9]+PolePar.fBlue_Mould-165-fDriverDDRActPos ))
			AND ( (aYellowPos[i9]+PolePar.fBlue_Mould-165-fDriverDDRActPos)<=PolePar.fPoleWidth+50 )AND aYellowPos[i9]>0 THEN						
			RecYRules[1]:=TRUE;//不纠偏
			EXIT;
		ELSE
				RecYRules[1]:=FALSE;//纠偏
		END_IF*)	
		IF      aYellowPos[i9]+PolePar.fBlue_Mould-fDriverDDRActPos<=165+80   AND   aYellowPos[i9]+PolePar.fBlue_Mould-fDriverDDRActPos>=165-80   
                        AND  aYellowPos[i9]>0   THEN
		        RecYRules[1]:=TRUE;//不纠偏
			EXIT;
		ELSE	
		        RecYRules[1]:=FALSE;//纠偏
		END_IF
		
	END_FOR	

										 
fbRectifyGM(
	bReset:=                      stSysState.bReset  ,  
	Execute:=                    RecY.bEnable  , 
	bCcw:=                       TRUE,//PolePar.Rec.bRectifyDir ,
	iRectifyMode:=           2 , //PolePar.Rec.iMode,
	bRecEn:=                   ,                         //纠偏容许条件
	fSensorActValue:=       stSenser.aiMouldRectifyBe , 
	fSensorActValue1:=     stSenser.aiMouldRectifyFr , 
	fSensorMaxValue:=     PolePar.Rec.fRecAxisPos_H, //从轴纠偏行程上限
	fSensorMinValue:=      PolePar.Rec.fRecAxisPos_L ,  //从轴纠偏行程下限
	fSensorBalanceValue:= PolePar.Rec.fRecBaseValue1+fArvTransverData2,//纠偏平衡位置
	fTolerance:=                PolePar.Rec.fRecBaseRange   ,  //纠偏死区                        , 
	fGMLengthSet:=           300, //纠偏距离标定
	fTimeAdjust:=                PolePar.Rec.fRectifyCoe , //纠偏时间标定
	bReady=>                    RecY.bReady ,
	bAutoRunning=>          RecY.bRecOK, 
	Error=> , 
	Axis_Rectify1:=         arrAxis[AxisNo.MouldRectify_Y] ,    
	Axis_VirGM:=        arrAxis[AxisNo.DriverDDR] ,    
	Axis_Time:=          arrAxis[NameNo.VirTimeWind] ,     );

RecY.bError:=fbRectifyGM.Error;//隔膜纠偏报警



(******************************************************************放卷纠偏，过程纠偏*****************************************************************************)
// 注意 : PoleWind代表过程纠偏      PoleProcess代表放卷纠偏   
//rMQUse[9](CLK:=stUwindTen.bError);//张力报警
//rMQUse[10](CLK:=stSysState.iMode=1);//自动
tonRecDelay(IN:= , PT:=T#300MS , Q=> , ET=> );


 //rtBoardPressTurn(CLK:=  stSysState.iMode=3  AND  ( arrCyCtrl[CYNo.BoardPressR].Io.DIOFFSwitch  OR  arrCyCtrl[CYNo.BoardPressL].Io.DIOFFSwitch ) , Q=> ); //检测压板有下压动作
 rtBoardPressTurn(CLK:= ((arrCyCtrl[NameNo.AnCYNo.Inflation_L].Status.OFFState AND PolePar.MQ.bWindSelect)OR (arrCyCtrl[NameNo.AnCYNo.Inflation_R].Status.OFFState   AND NOT PolePar.MQ.bWindSelect) ) , Q=> ); //检测压板有下压动作
 rtBreakError(CLK:= stUwindTen.bError AND  ((stAuxDriverTen.fDanserDegree>PolePar.MQ.AuxDriverTenMaxPos-2)  OR  (stAuxDriverTen.fDanserDegree<PolePar.MQ.AuxDriverTenMinPos+2))   , Q=> ); //检测到断带
       IF   rtBoardPressTurn.Q OR rtBreakError.Q THEN
		    fCyDDRActPos:=fDriverDDRActPos;//记录主驱当前位置
			bCyDDRMark:=TRUE;//滞后纠偏标志
	   END_IF
  IF  bCyDDRMark  AND    fDriverDDRActPos-fCyDDRActPos >=2500     THEN  //料带走2500mm后恢复纠偏
       bCyDDRMark:=FALSE;//滞后纠偏标志复位
  END_IF
	IF  bCyDDRMark  AND    fDriverDDRActPos < fCyDDRActPos-2500     THEN  //主驱位置小于主驱记录位置，复位滞后纠偏
		bCyDDRMark:=FALSE;//滞后纠偏标志复位
	END_IF
	
 // rtRecManual1(CLK:=  stSysState.iMode=3 AND   arrAxis[VirAxisNo.VirMain].NcToPlc.SetVelo=0            , Q=> );  //手动状态
//  rtRecManual1(CLK:=   arrAxis[VirAxisNo.VirMain].NcToPlc.SetVelo=0            , Q=> );  //手动状态
  tonRecCenterDelay(IN:= , PT:=T#4.5S , Q=> , ET=> );  //居中移动延时
  
 
  CASE  RecSetp  OF
	    0:  //检查是否是处于手动状态
          tonRecDelay.IN:=FALSE;
          tonRecCenterDelay.IN:=FALSE;
          RecSetp:=1;
  
	  1:  //检查是否是处于手动状态
	       tonRecDelay.IN:=TRUE;
		   IF  tonRecDelay.Q THEN
			    IF (  (stSysState.iMode=3 AND   arrAxis[VirAxisNo.VirMain].NcToPlc.SetVelo=0)   OR 
                     stUwindTen.bError   OR
                     bCyDDRMark    )   AND     iRecStatus<>1     THEN// AND     iRecStatus<>1  
			         bFlgRecManual:=TRUE; 
		        END_IF
			    tonRecDelay.IN:=FALSE;
	           RecSetp:=2;
		   END_IF
	  2:  //纠偏居中
	       tonRecDelay.IN:=TRUE;
		   
	      IF stSysState.iMode=3    AND  (  (fbRotateSwitchCode.iCodeOut=11 OR fbRotateSwitchCode.iCodeOut=3)   AND rtPoleBtn.Q     )    THEN  //AND   iRecStatus<>3  
	            tonRecCenterDelay.IN:=TRUE;
				bFlgRecCenter:=TRUE;
			    bRecCenterMoving:=TRUE;
		  END_IF
		  
		  IF  bRecCenterMoving THEN
			    IF  tonRecCenterDelay.Q THEN
				     bRecCenterMoving:=FALSE;
					  tonRecCenterDelay.IN:=FALSE;
					   tonRecDelay.IN:=FALSE;
                     RecSetp:=3;	  		 
			   END_IF
		  ELSE  
			  IF  tonRecDelay.Q THEN
				   tonRecDelay.IN:=FALSE;
			      tonRecCenterDelay.IN:=FALSE;
			      RecSetp:=3;	  
		  	 END_IF		
		  END_IF
		   
	3:  //纠偏自动启动
	      tonRecDelay.IN:=TRUE;
		    IF  tonRecDelay.Q THEN
			     IF    stSysState.iMode=1 AND  stUwindTen.bTensionOK   AND   NOT  bCyDDRMark     THEN  // AND   iRecStatus<>2
			            bFlgRecAuto:=TRUE; 
		          END_IF		
				 tonRecDelay.IN:=FALSE;
	            RecSetp:=0;	   
		   END_IF
		   
  END_CASE
  
  
  
  IF  bFlgRecManual THEN
	  	arrRecCtrl[RecNo.PoleWind].Cmd.bCentre:=FALSE;
		arrRecCtrl[RecNo.PoleWind].Cmd.bAuto :=FALSE;
		//arrRecCtrl[RecNo.PoleWind].Cmd.bLock:=FALSE;
		arrRecCtrl[RecNo.PoleWind].Cmd.bManual:=TRUE;
		
		arrRecCtrl[RecNo.PoleProcess].Cmd.bCentre:=FALSE;
		arrRecCtrl[RecNo.PoleProcess].Cmd.bAuto :=FALSE;
	//	arrRecCtrl[RecNo.PoleProcess].Cmd.bLock:=FALSE;
		arrRecCtrl[RecNo.PoleProcess].Cmd.bManual:=TRUE;
		
		iRecStatus:=1;
		bFlgRecManual:=FALSE;
  END_IF
  
  
    IF  bFlgRecAuto THEN
	  	arrRecCtrl[RecNo.PoleWind].Cmd.bCentre:=FALSE;
		arrRecCtrl[RecNo.PoleWind].Cmd.bAuto :=TRUE;
		//arrRecCtrl[RecNo.PoleWind].Cmd.bLock:=FALSE;
		arrRecCtrl[RecNo.PoleWind].Cmd.bManual:=FALSE;
		
		arrRecCtrl[RecNo.PoleProcess].Cmd.bCentre:=FALSE;
		arrRecCtrl[RecNo.PoleProcess].Cmd.bAuto :=TRUE;
		//arrRecCtrl[RecNo.PoleProcess].Cmd.bLock:=FALSE;
		arrRecCtrl[RecNo.PoleProcess].Cmd.bManual:=FALSE;
		iRecStatus:=2;
		bFlgRecAuto:=FALSE;
  END_IF

  
   IF  bFlgRecCenter THEN
	  //	arrRecCtrl[RecNo.PoleWind].Cmd.bCentre:=TRUE;
		//arrRecCtrl[RecNo.PoleWind].Cmd.bAuto :=FALSE;
		//arrRecCtrl[RecNo.PoleWind].Cmd.bLock:=FALSE;
		//arrRecCtrl[RecNo.PoleWind].Cmd.bManual:=FALSE;
		
		arrRecCtrl[RecNo.PoleProcess].Cmd.bCentre:=TRUE;
		arrRecCtrl[RecNo.PoleProcess].Cmd.bAuto :=FALSE;
		//arrRecCtrl[RecNo.PoleProcess].Cmd.bLock:=FALSE;
		arrRecCtrl[RecNo.PoleProcess].Cmd.bManual:=FALSE;
		iRecStatus:=3;
		bFlgRecCenter:=FALSE;
  END_IF
  
  
 (* 
 	5:  //纠偏自动锁定
	      IF    stSysState.iMode=1   THEN
			     arrRecCtrl[RecNo.PoleWind].Cmd.bLock:=TRUE;
				 arrRecCtrl[RecNo.PoleProcess].Cmd.bLock:=TRUE;
		ELSE		 
			     arrRecCtrl[RecNo.PoleWind].Cmd.bLock:=FALSE;
				 arrRecCtrl[RecNo.PoleProcess].Cmd.bLock:=FALSE;	 	 
		  END_IF
		  
	     RecSetp:=0;	 
*)


(*

  CASE  RecSetp  OF
	    0:  //检查是否是处于手动状态
          tonRecDelay.IN:=FALSE;
          tonRecCenterDelay.IN:=FALSE;
          RecSetp:=1;
  
	  1:  //检查是否是处于手动状态
	       tonRecDelay.IN:=TRUE;
	      IF (  (stSysState.iMode=3 AND   arrAxis[VirAxisNo.VirMain].NcToPlc.SetVelo=0)   OR 
                stUwindTen.bError   OR
                bCyDDRMark    ) THEN// AND     iRecStatus<>1  
			    bFlgRecManual:=TRUE; 
		   END_IF
		   IF  tonRecDelay.Q THEN
			    tonRecDelay.IN:=FALSE;
	           RecSetp:=2;
		   END_IF
	  2:  //纠偏居中
	       tonRecDelay.IN:=TRUE;
		   
	      IF stSysState.iMode=3    AND  (  (fbRotateSwitchCode.iCodeOut=11 OR fbRotateSwitchCode.iCodeOut=3)   AND rtPoleBtn.Q     )    THEN  //AND   iRecStatus<>3  
	            tonRecCenterDelay.IN:=TRUE;
				bFlgRecCenter:=TRUE;
			    bRecCenterMoving:=TRUE;
		  END_IF
		  
		  IF  bRecCenterMoving THEN
			    IF  tonRecCenterDelay.Q THEN
				     bRecCenterMoving:=FALSE;
					  tonRecCenterDelay.IN:=FALSE;
					   tonRecDelay.IN:=FALSE;
                     RecSetp:=3;	  		 
			   END_IF
		  ELSE  
			  IF  tonRecDelay.Q THEN
				   tonRecDelay.IN:=FALSE;
			      tonRecCenterDelay.IN:=FALSE;
			      RecSetp:=3;	  
		  	 END_IF		
		  END_IF
		   
	3:  //纠偏自动启动
	      tonRecDelay.IN:=TRUE;
	      IF    stSysState.iMode=1 AND  stUwindTen.bTensionOK   AND   NOT  bCyDDRMark     THEN  // AND   iRecStatus<>2
			  bFlgRecAuto:=TRUE; 
		  END_IF
		    IF  tonRecDelay.Q THEN
				 tonRecDelay.IN:=FALSE;
	            RecSetp:=0;	   
		   END_IF
		   
  END_CASE

*)
















(*
//////////////////////////////////模具Y纠偏//////////////////////////////////
	IF arrAxisCtrl[VirAxisNo.VirMain].Status.fModuloSetPos>=20  AND arrAxisCtrl[VirAxisNo.VirMain].Status.fModuloSetPos<250 AND
	   arrAxisCtrl[VirAxisNo.VirMain].Status.Moving AND  stDriverCam.bInSync  AND NOT ProductPar.iModeEN.bMouldYRecEN AND NOT RecYRules[1] THEN
		RecY.bEnable:=TRUE;				
	ELSE
		RecY.bEnable:=FALSE;	
	END_IF


//黄标不纠偏范围判断,,,-170指黄标感应器高裁切距离-170=黄标感应器到纠偏传感器的距离,,,即纠偏传感器到裁切切刀距离为170
	FOR i9:=20 TO 1 BY -1 DO	
		IF (PolePar.fPoleWidth-35<=(aYellowPos[i9]+PolePar.fBlue_Mould+5*PolePar.fPoleWidth-170-fDriverDDRActPos ))
			AND ( (aYellowPos[i9]+PolePar.fBlue_Mould+5*PolePar.fPoleWidth-170-fDriverDDRActPos)<=PolePar.fPoleWidth+35 )
			AND aYellowPos[i9]>0 THEN						
				RecYRules[1]:=TRUE;//不纠偏
				EXIT;
		ELSE
				RecYRules[1]:=FALSE;//纠偏
		END_IF
	END_FOR	
	
	
	
	
	
fbTailCurl(
	Enable:=RecY.bEnable , 
	RestHMI:=stSysState.bReset , 
	MasterNo:=NameNo.VirTimeWind , 
	SlaveNo:=AxisNo.MouldRectify_Y , 
	MasterValue:=arrAxisCtrl[NameNo.VirTimeWind].Status.fActVelo , 
	RecDevEqupos1:=PolePar.Rec.fRecBaseValue1,//SEL(CCD_Rounde.CWW,PolePar.Rec.fRecBaseValue1+CCD_Rounde.ResultData,PolePar.Rec.fRecBaseValue1-CCD_Rounde.ResultData)  , 
	RecDevEqupos2:=PolePar.Rec.fRecBaseValue2 , 
	RecDevValueSet:=PolePar.Rec.fRecBaseRange , 
	RecDevPV1:=stSenser.aiMouldRectifyBe , 
	RecDevPV2:=stSenser.aiMouldRectifyFr , 
	RecDevSpeedCoe:=PolePar.Rec.fRectifyCoe , 
	CWW:=PolePar.Rec.bRectifyDir , 
	AxisintiPos:=arrAxisPar[AxisNo.MouldRectify_Y].arrTargetPoint[1] , 
	AxisPos_H:=PolePar.Rec.fRecAxisPos_H , 
	AxisPos_L:=PolePar.Rec.fRecAxisPos_L , 
	bMode:=PolePar.Rec.iMode,
	iMainVel := PolePar.iMainVel , 
	bError=>RecY.bError , 
	bRecOK=>RecY.bRecOK , 
	bReady=>RecY.bReady );
	PolePar.Rec.iMode:=1;



//CCD闭环补偿
CCD_Rounde(
	CCD_Enable:=CCD_Rounde.CCD_Enable , //启动
	CWW:= , //纠偏方向选择
	IntervalNum:=PolePar.IntervalNum , //片间距
	KI_Riao:=PolePar.KI_Riao , //比例系数
	Databace_R3:=PolePar.Databace_R3  , //CCD 非极耳侧纵深基准正极5.6  负极2.6
	Databace_R4:=PolePar.Databace_R4 , //CCD 极耳侧纵深基准正极5.6  负极2.6
	CCD_RoundedSize_R3:=CCD_COM.Size.RoundedSize1 , //CCD 非极耳侧纵深
	CCD_RoundedSize_R4:=CCD_COM.Size.RoundedSize2 , //CCD 极耳侧纵深
	Limt_Max:=PolePar.Limt_Max , //最大补偿值
	Limt_Min:=PolePar.Limt_Min, //最小补偿值
	JzData:=PolePar.Rec.fRecBaseValue1,
	ResultData=> );//补偿值输出
CCD_Rounde.KK;//启动开关；
*)


(*

IF stSysState.iMode=1 THEN
	IF (fCyDDRActPos+2900-fDriverDDRActPos<=0  ) AND NOT bCyDDRMark THEN
		bCyDDRMark:=TRUE;//设备自动时纠偏启动标志位
		arrRecCtrl[RecNo.PoleWind].Cmd.bCentre:=FALSE;
		arrRecCtrl[RecNo.PoleWind].Cmd.bAuto :=TRUE;
		arrRecCtrl[RecNo.PoleWind].Cmd.bLock:=FALSE;
		arrRecCtrl[RecNo.PoleWind].Cmd.bManual:=FALSE;
		
		arrRecCtrl[RecNo.PoleProcess].Cmd.bCentre:=FALSE;
		arrRecCtrl[RecNo.PoleProcess].Cmd.bAuto :=TRUE;
		arrRecCtrl[RecNo.PoleProcess].Cmd.bLock:=FALSE;
		arrRecCtrl[RecNo.PoleProcess].Cmd.bManual:=FALSE;
	END_IF
END_IF



//张力报警放卷剪片、行进纠偏回手动
IF rMQUse[9].Q THEN
	arrRecCtrl[RecNo.PoleWind].Cmd.bCentre:=FALSE;
	arrRecCtrl[RecNo.PoleWind].Cmd.bAuto :=FALSE;
	arrRecCtrl[RecNo.PoleWind].Cmd.bLock:=FALSE;
	arrRecCtrl[RecNo.PoleWind].Cmd.bManual:=TRUE;
	
	arrRecCtrl[RecNo.PoleProcess].Cmd.bCentre:=FALSE;
	arrRecCtrl[RecNo.PoleProcess].Cmd.bAuto :=FALSE;
	arrRecCtrl[RecNo.PoleProcess].Cmd.bLock:=FALSE;
	arrRecCtrl[RecNo.PoleProcess].Cmd.bManual:=TRUE;
END_IF


//气涨轴松开时放卷纠偏居中	
IF PolePar.MQ.bWindSelect THEN
	IF rMQUse[7].Q THEN	
		arrRecCtrl[RecNo.PoleProcess].Cmd.bCentre:=FALSE;
		arrRecCtrl[RecNo.PoleProcess].Cmd.bAuto :=TRUE;
		arrRecCtrl[RecNo.PoleProcess].Cmd.bLock:=FALSE;
		arrRecCtrl[RecNo.PoleProcess].Cmd.bManual:=FALSE;
	END_IF
	IF fMQUse[7].Q THEN	
		arrRecCtrl[RecNo.PoleProcess].Cmd.bCentre:=TRUE;
		arrRecCtrl[RecNo.PoleProcess].Cmd.bAuto :=FALSE;
		arrRecCtrl[RecNo.PoleProcess].Cmd.bLock:=FALSE;
		arrRecCtrl[RecNo.PoleProcess].Cmd.bManual:=FALSE;
	END_IF
ELSE	
	IF rMQUse[8].Q THEN	
		arrRecCtrl[RecNo.PoleProcess].Cmd.bCentre:=FALSE;
		arrRecCtrl[RecNo.PoleProcess].Cmd.bAuto :=TRUE;
		arrRecCtrl[RecNo.PoleProcess].Cmd.bLock:=FALSE;
		arrRecCtrl[RecNo.PoleProcess].Cmd.bManual:=FALSE;
	END_IF
	IF fMQUse[8].Q THEN	
		arrRecCtrl[RecNo.PoleProcess].Cmd.bCentre:=TRUE;
		arrRecCtrl[RecNo.PoleProcess].Cmd.bAuto :=FALSE;
		arrRecCtrl[RecNo.PoleProcess].Cmd.bLock:=FALSE;
		arrRecCtrl[RecNo.PoleProcess].Cmd.bManual:=FALSE;
	END_IF
END_IF

*)
END_ACTION

ACTION F07Condition:
MQ_alarm_ton[1](PT:=T#100MS);
MQ_alarm_ton[2](PT:=T#100MS);
MQ_alarm_ton[3](PT:=T#100MS);
MQ_alarm_ton[4](PT:=T#100MS);
MQ_alarm_ton[5](PT:=T#100MS);
MQ_alarm_ton[6](PT:=T#100MS);
MQ_alarm_ton[7](PT:=T#100MS);
MQ_alarm_ton[8](PT:=T#100MS);
MQ_alarm_ton[9](PT:=T#100MS);
MQ_alarm_ton[10](PT:=T#100MS);
MQ_alarm_ton[11](PT:=T#100MS);
MQ_alarm_ton[12](PT:=T#100MS);
MQ_alarm_ton[13](PT:=T#100MS);
MQ_alarm_ton[14](PT:=T#100MS);
MQ_alarm_ton[15](PT:=T#100MS);
MQ_alarm_ton[16](PT:=T#100MS);
MQ_alarm_ton[17](PT:=T#100MS);





////////////////////////////////////线扫IO触发////////////////////////////////////////
rLineScanOK_UP(CLK:=stSenser.bLineScanResult1_UP , Q=> );
rLineScanNG_UP(CLK:=stSenser.bLineScanResult2_UP , Q=> );
rLineScanOK_Down(CLK:=stSenser.bLineScanResult1_Down , Q=> );
rLineScanNG_Down(CLK:=stSenser.bLineScanResult2_Down , Q=> );
IF rLineScanOK_UP.Q THEN
	bLineScanResult1_UP:=TRUE;
END_IF
IF rLineScanNG_UP.Q THEN
	bLineScanResult2_UP:=TRUE;
END_IF
IF rLineScanOK_Down.Q THEN
	bLineScanResult1_Down:=TRUE;
END_IF
IF rLineScanNG_Down.Q THEN
	bLineScanResult2_Down:=TRUE;
END_IF


////////////////////////////////////微分&延时////////////////////////////////////
rtbtnRest(CLK:=stSysState.bReset , Q=> );
rtCondition[1](CLK:=bTest[1],Q=>);//测试1
tonCondition[1](In:=CCD_Com.bLineHeart,PT:=T#2S);//线扫软件心跳延时1
tonCondition[2](In:=NOT CCD_Com.bLineHeart,PT:=T#2S);//线扫软件心跳延时2
tonCondition[3](In:=CCD_Com.bAreaHeart,PT:=T#2S);//面阵软件心跳延时1
tonCondition[4](In:=NOT CCD_Com.bAreaHeart,PT:=T#2S);//面阵软件心跳延时2

tonCondition[5](In:=arrRecCtrl[RecNo.PoleWind].Cmd.bCentre,PT:=T#120MS);//放卷纠偏触发回中延时
tonCondition[6](In:=arrRecCtrl[RecNo.PoleWind].Cmd.bAuto,PT:=T#120MS);//放卷纠偏触发自动延时
tonCondition[7](In:=arrRecCtrl[RecNo.PoleWind].Cmd.bManual,PT:=T#120MS);//放卷纠偏触发手动延时
tonCondition[8](In:=arrRecCtrl[RecNo.PoleProcess].Cmd.bCentre,PT:=T#120MS);//过程纠偏触发回中延时
tonCondition[9](In:=arrRecCtrl[RecNo.PoleProcess].Cmd.bAuto,PT:=T#120MS);//过程纠偏触发自动延时
tonCondition[10](In:=arrRecCtrl[RecNo.PoleProcess].Cmd.bManual,PT:=T#120MS);//过程纠偏触发手动延时v


////////////////////////////////////////////自动运行准备好条件//////////////////////////////////
IF ((stUwindTen.bTensionOK AND  PolePar.MQ.bWindSelect) OR(stUwindTen.bTensionOK AND NOT  PolePar.MQ.bWindSelect))  THEN
	bAutoReadyTemp1:=TRUE;//张力准备好
ELSE
	bAutoReadyTemp1:=FALSE;
END_IF															
IF stPoleBufferCam.bCreatTableDone AND stDriverCam.bCreatTableDone AND stCuterCam.bCreatTableDone AND 
	stVirBeltCam.bCreatTableDone (*AND stNGPushCam.bCreatTableDone*) AND stMouldCam.bCreatTableDone AND
	stCCDPressCam.bCreatTableDone THEN
	bAutoReadyTemp2:=TRUE;	//凸轮创建OK
ELSE
	bAutoReadyTemp2:=FALSE;
END_IF	
IF 	arrCyCtrl[CYNo.DriverPressDDR].Status.ONState  THEN
	bAutoReadyTemp3:=TRUE;		//气缸准备OK
ELSE
	bAutoReadyTemp3:=FALSE;
END_IF

IF arrAxisCtrl[AxisNo.Mould].Status.Enabled AND arrAxisCtrl[AxisNo.MouldRectify_X].Status.Enabled AND arrAxisCtrl[AxisNo.MouldRectify_Y].Status.Enabled AND 
	arrAxisCtrl[AxisNo.Cuter].Status.Enabled AND arrAxisCtrl[AxisNo.CuterDegRectify].Status.Enabled AND arrAxisCtrl[AxisNo.CuterBeltChange].Status.Enabled AND
	(*arrAxisCtrl[AxisNo.NGPush1].Status.Enabled AND arrAxisCtrl[AxisNo.NGPush2].Status.Enabled AND *)arrAxisCtrl[AxisNo.CCDPressPush].Status.Enabled AND
	arrAxisCtrl[AxisNo.UnWind_L].Status.Enabled AND arrAxisCtrl[AxisNo.UnWind_R].Status.Enabled (*AND arrAxisCtrl[AxisNo.DriverAux].Status.Enabled *)AND
	arrAxisCtrl[AxisNo.DriverDDR].Status.Enabled AND arrAxisCtrl[AxisNo.BuffeLine].Status.Enabled AND arrAxisCtrl[AxisNo.CuterBelt].Status.Enabled AND 
	arrAxisCtrl[AxisNo.NGPushReverseBelt].Status.Enabled AND arrAxisCtrl[AxisNo.DedustBelt].Status.Enabled AND arrAxisCtrl[AxisNo.DedustReverseBelt].Status.Enabled AND 
	arrAxisCtrl[AxisNo.SubBelt1].Status.Enabled AND arrAxisCtrl[AxisNo.SubBelt2].Status.Enabled AND arrAxisCtrl[AxisNo.SubBelt3].Status.Enabled AND
	arrAxisCtrl[VirAxisNo.VirBelt].Status.Enabled AND arrAxisCtrl[VirAxisNo.VirDriver].Status.Enabled AND arrAxisCtrl[VirAxisNo.VirMain].Status.Enabled THEN
	bAutoReadyTemp4:=TRUE;		//轴准备OK
ELSE
	bAutoReadyTemp4:=FALSE;
END_IF

IF NOT arrAxisCtrl[AxisNo.Mould].Status.Error AND NOT arrAxisCtrl[AxisNo.Mould] .Status.ErrorLimitSwitch AND  
	NOT arrAxisCtrl[AxisNo.MouldRectify_X].Status.Error AND NOT arrAxisCtrl[AxisNo.MouldRectify_X] .Status.ErrorLimitSwitch AND  
	NOT arrAxisCtrl[AxisNo.MouldRectify_Y].Status.Error AND NOT arrAxisCtrl[AxisNo.MouldRectify_Y] .Status.ErrorLimitSwitch AND  
	NOT arrAxisCtrl[AxisNo.Cuter].Status.Error AND NOT arrAxisCtrl[AxisNo.Cuter] .Status.ErrorLimitSwitch AND 
	NOT arrAxisCtrl[AxisNo.CuterDegRectify].Status.Error AND NOT arrAxisCtrl[AxisNo.CuterDegRectify] .Status.ErrorLimitSwitch AND  	
	NOT arrAxisCtrl[AxisNo.CuterBeltChange].Status.Error AND NOT arrAxisCtrl[AxisNo.CuterBeltChange] .Status.ErrorLimitSwitch AND  
	NOT arrAxisCtrl[AxisNo.CCDPressPush].Status.Error AND NOT arrAxisCtrl[AxisNo.CCDPressPush] .Status.ErrorLimitSwitch AND   
	NOT arrAxisCtrl[AxisNo.UnWind_L].Status.Error AND NOT arrAxisCtrl[AxisNo.UnWind_L] .Status.ErrorLimitSwitch AND   
	NOT arrAxisCtrl[AxisNo.UnWind_R].Status.Error AND NOT arrAxisCtrl[AxisNo.UnWind_R] .Status.ErrorLimitSwitch AND   
	NOT arrAxisCtrl[AxisNo.DriverDDR].Status.Error AND NOT arrAxisCtrl[AxisNo.DriverDDR] .Status.ErrorLimitSwitch AND   
	NOT arrAxisCtrl[AxisNo.BuffeLine].Status.Error AND NOT arrAxisCtrl[AxisNo.BuffeLine] .Status.ErrorLimitSwitch AND    
	NOT arrAxisCtrl[AxisNo.CuterBelt].Status.Error AND NOT arrAxisCtrl[AxisNo.CuterBelt] .Status.ErrorLimitSwitch AND   
	NOT arrAxisCtrl[AxisNo.NGPushReverseBelt].Status.Error AND NOT arrAxisCtrl[AxisNo.NGPushReverseBelt] .Status.ErrorLimitSwitch AND    
	NOT arrAxisCtrl[AxisNo.DedustBelt].Status.Error AND NOT arrAxisCtrl[AxisNo.DedustBelt] .Status.ErrorLimitSwitch AND    
	NOT arrAxisCtrl[AxisNo.DedustReverseBelt].Status.Error AND NOT arrAxisCtrl[AxisNo.DedustReverseBelt] .Status.ErrorLimitSwitch AND     
	NOT arrAxisCtrl[AxisNo.SubBelt1].Status.Error AND NOT arrAxisCtrl[AxisNo.SubBelt1] .Status.ErrorLimitSwitch AND    
	NOT arrAxisCtrl[AxisNo.SubBelt2].Status.Error AND NOT arrAxisCtrl[AxisNo.SubBelt2] .Status.ErrorLimitSwitch AND    
	NOT arrAxisCtrl[AxisNo.SubBelt3].Status.Error AND NOT arrAxisCtrl[AxisNo.SubBelt3] .Status.ErrorLimitSwitch AND    
	NOT arrAxisCtrl[VirAxisNo.VirBelt].Status.Error AND NOT arrAxisCtrl[VirAxisNo.VirBelt] .Status.ErrorLimitSwitch AND   
	NOT arrAxisCtrl[VirAxisNo.VirDriver].Status.Error AND NOT arrAxisCtrl[VirAxisNo.VirDriver] .Status.ErrorLimitSwitch AND    
	NOT arrAxisCtrl[VirAxisNo.VirMain].Status.Error AND NOT arrAxisCtrl[VirAxisNo.VirMain] .Status.ErrorLimitSwitch THEN
		bAutoReadyTemp5:=TRUE;
ELSE
	bAutoReadyTemp5:=FALSE;
END_IF

IF 	bAutoReadyTemp2 AND NOT SysPart.bErrorStop AND SysPart.Homed AND bAutoReadyTemp4 AND bAutoReadyTemp5 THEN
	SysPart.bAutoCondition1:=TRUE;
ELSE
	SysPart.bAutoCondition1:=FALSE;		
END_IF
IF 	bAutoReadyTemp2 AND NOT SysPart.bErrorStop AND SysPart.Homed AND (ProductPar.iModeEN.bEmptyRunEN OR bAutoReadyTemp1 AND bAutoReadyTemp3 ) THEN
	SysPart.bAutoCondition2:=TRUE;
ELSE
	SysPart.bAutoCondition2:=FALSE;		
END_IF 


//新黄标、接带检测------------------------新
		PolePar.fLugBreadth;//极耳宽度
		PolePar.fCutBreadth;//极耳边到切刀切点宽度
		PolePar.fYellowBreadth;//黄标宽度
		//黄标第一片到R角距离5片，，，到裁切5片共10片，，，到踢废n片
ftAuto[1](CLK:=stSenser.bYellowCheck_C , Q=> );//黄标检测下降沿
ftAuto[2](CLK:=stSenser.biTabHave , Q=> );//极耳检测下降沿			
	//假设黄标感应器在第一片与第二片之间	
	IF arrAxisCtrl[VirAxisNo.VirMain].Status.fModuloActPos>=0 AND arrAxisCtrl[VirAxisNo.VirMain].Status.fModuloActPos<=260 AND arrAxisCtrl[VirAxisNo.VirMain].Status.Moving THEN
		IF NOT bLugActPosMark_f THEN		
			IF rtAuto[11].Q THEN
				fLugActPos:=arrAxisCtrl[AxisNo.DriverDDR].Status.fActPos;//极耳位置记录---------------P1
				bLugActPosMark_r:=TRUE;//上升沿极耳位置已记录标志位
			END_IF			
		END_IF
		IF NOT  bLugActPosMark_r THEN
			IF ftAuto[2].Q THEN
				fLugActPos:=arrAxisCtrl[AxisNo.DriverDDR].Status.fActPos-50;//极耳位置记录-----------------P1
				bLugActPosMark_f:=TRUE;//下降沿极耳位置已记录标志位
			END_IF
		END_IF
	//黄标位置记录
		IF 	rtAuto[10].Q  THEN//----黄标只取上升沿
			bYellowActPosMark:=TRUE;//黄标位置已记录标志位
			fYellowMarkActPos:=arrAxisCtrl[AxisNo.DriverDDR].Status.fActPos;//黄标位置记录	------------P2
		END_IF
	ELSIF arrAxisCtrl[VirAxisNo.VirMain].Status.fModuloActPos>270 AND arrAxisCtrl[VirAxisNo.VirMain].Status.fModuloActPos<300 THEN//-----------数据移位已经完成			
		IF bYellowActPosMark AND ( bLugActPosMark_r OR bLugActPosMark_f)  THEN//------------黄标有感应到，极耳有感应到		
			rYellowPosRel:=fYellowMarkActPos-fLugActPos;//黄标感应器相对于极耳位置的差-----------------------S黄标
			rYellowJumpPos1:=PolePar.fCutBreadth-PolePar.fYellowBreadth;//黄标跳切区间判断位置1-------------S1
			rYellowJumpPos2:=PolePar.fCutBreadth+PolePar.fYellowBreadth;//黄标跳切区间判断位置2------------S2							
			IF rYellowPosRel<0 THEN//黄标在极耳左侧---不跳切						
				bYellowMark[2]:=TRUE;//---------黄标在2#片
			ELSE//黄标在极耳右侧
				IF rYellowPosRel<rYellowJumpPos1 THEN//------------------------不跳切
					bYellowMark[2]:=TRUE;	//-------------黄标在2#片
				ELSIF rYellowPosRel>rYellowJumpPos2 THEN//---------------------不跳切
					bYellowMark[1]:=TRUE;	//-------------黄标在1#片
				ELSE//--------------黄标在极片1和极片2切刀位置
					bYellowMark[1]:=TRUE;	//-------------黄标在1#片		
					bYellowMark[2]:=TRUE;//	-------------黄标在2#片		
				END_IF
			END_IF
		ELSIF  bYellowActPosMark AND NOT bLugActPosMark_r AND NOT bLugActPosMark_f THEN //--------------黄标有感应到，极耳没有感应到
			bYellowMark[1]:=TRUE;	//-------------黄标在1#片		
			bYellowMark[2]:=TRUE;	//-------------黄标在2#片		
		ELSIF NOT bYellowActPosMark AND ( bLugActPosMark_r OR bLugActPosMark_f ) THEN//-------------------极耳有感应到，黄标没感应到，，正常片
			bLugActPosMark_r:=FALSE;//上升沿极耳位置已记录标志位
			bLugActPosMark_f:=FALSE;//下降沿极耳位置已记录标志位
			bYellowActPosMark:=FALSE;//黄标位置已记录标志位
			fLugActPos:=0;
			fYellowMarkActPos:=0;
			rYellowPosRel:=0;//黄标感应器相对于极耳位置的差
			rYellowJumpPos1:=0;//黄标跳切区间判断位置1
			rYellowJumpPos2:=0;//黄标跳切区间判断位置2
		ELSE//-----------黄标和极耳都没感应到
			bYellowMark[1]:=TRUE;	//-------------黄标在1#片		
			bYellowMark[2]:=TRUE;	//-------------黄标在2#片		
		END_IF
	ELSIF arrAxisCtrl[VirAxisNo.VirMain].Status.fModuloActPos>300 AND arrAxisCtrl[VirAxisNo.VirMain].Status.fModuloActPos<350 THEN//
		bLugActPosMark_r:=FALSE;//上升沿极耳位置已记录标志位
		bLugActPosMark_f:=FALSE;//下降沿极耳位置已记录标志位
		bYellowActPosMark:=FALSE;//黄标位置已记录标志位
		fLugActPos:=0;
		fYellowMarkActPos:=0;
		rYellowPosRel:=0;//黄标感应器相对于极耳位置的差
		rYellowJumpPos1:=0;//黄标跳切区间判断位置1
		rYellowJumpPos2:=0;//黄标跳切区间判断位置2
	END_IF
		
		
		
		
		
		
		

(*
//////////////裁切前黄标检测//////////-------------------原版
IF arrAxisCtrl[VirAxisNo.VirMain].Status.fModuloActPos>=0 AND arrAxisCtrl[VirAxisNo.VirMain].Status.fModuloActPos<260 AND
	arrAxisCtrl[VirAxisNo.VirMain].Status.Moving AND NOT stSenser.bYellowCheck_C  THEN
	YellowmarkNG[1]:=0;//裁切前黄标NG
END_IF
*)




		(*IF stUwindLTen.fWindDiameter<PolePar.fDiameterWarn_L AND PolePar.fDiameterWarn_L>0 THEN
			stAlarm.arrLightWarn[14]:=TRUE;//左极片料卷即将用完！
		END_IF
		IF stUwindLTen.fWindDiameter<PolePar.fDiameterAlarm_L AND PolePar.fDiameterAlarm_L>0 THEN
			stAlarm.arrFlowAlarm[15]:=TRUE;//左极片料卷已用完，请停机处理！
		END_IF	
	
		IF stUwindRTen.fWindDiameter<PolePar.fDiameterWarn_R AND PolePar.fDiameterWarn_R>0 THEN
			stAlarm.arrLightWarn[15]:=TRUE;
		END_IF
		IF stUwindRTen.fWindDiameter<PolePar.fDiameterAlarm_R AND PolePar.fDiameterAlarm_R>0 THEN
			stAlarm.arrFlowAlarm[16]:=TRUE;//右极片料卷已用完，请停机处理！
		END_IF*)


(*/////////卷径报警&警告/////////
IF NOT ProductPar.iModeEN.bEmptyRunEN THEN
	IF PolePar.MQ.bWindSelect THEN
		IF stUwindLTen.fWindDiameter<PolePar.fDiameterWarn_L AND PolePar.fDiameterWarn_L>0 THEN
			stAlarm.arrLightWarn[14]:=TRUE;//左极片料卷即将用完！
		END_IF
		IF stUwindLTen.fWindDiameter<PolePar.fDiameterAlarm_L AND PolePar.fDiameterAlarm_L>0 THEN
			stAlarm.arrFlowAlarm[15]:=TRUE;//左极片料卷已用完，请停机处理！
		END_IF	
	ELSE	
		IF stUwindRTen.fWindDiameter<PolePar.fDiameterWarn_R AND PolePar.fDiameterWarn_R>0 THEN
			stAlarm.arrLightWarn[15]:=TRUE;//右极片料卷即将用完！
		END_IF
		IF stUwindRTen.fWindDiameter<PolePar.fDiameterAlarm_R AND PolePar.fDiameterAlarm_R>0 THEN
			stAlarm.arrFlowAlarm[16]:=TRUE;//右极片料卷已用完，请停机处理！
		END_IF
	END_IF
END_IF*)

//////////////////////////////////偏心轮类电机处理//////////////////////////////////
//////////////冲R角模具////////////
FOR i2:=0 TO 10 BY 1 DO			
	IF arrAxisCtrl[AxisNo.Mould].Cmd.arrbModuloGo[i2] AND arrAxis[AxisNo.Mould].Status.StandStill THEN		
		IF NOT arrAxisCtrl[AxisNo.Mould].Cmd.arrbModuloPoint[i2] THEN	
			arrAxisCtrl[AxisNo.Mould].Cmd.fPositon_of_Mod:=arrAxisPar[AxisNo.Mould].arrTargetPoint[i2];//绝对模长位置定位
			arrAxisCtrl[AxisNo.Mould].Cmd.bMoveModulo:=TRUE;
			arrAxisCtrl[AxisNo.Mould].Cmd.arrbModuloGo[i2]:=FALSE;
		ELSE	
			arrAxisCtrl[AxisNo.Mould].Cmd.arrbModuloGo[i2]:=FALSE;
		END_IF	
	END_IF		
	IF arrAxisPar[AxisNo.Mould].arrTargetPoint[i2]-0.1<= arrAxisCtrl[AxisNo.Mould].Status.fModuloActPos AND		
		arrAxisPar[AxisNo.Mould].arrTargetPoint[i2]+0.1>=arrAxisCtrl[AxisNo.Mould].Status.fModuloActPos AND	
		NOT arrAxisCtrl[AxisNo.Mould].Cmd.bMoveModulo THEN	
		arrAxisCtrl[AxisNo.Mould].Cmd.arrbModuloPoint[i2]:=TRUE;	
	ELSE		
		arrAxisCtrl[AxisNo.Mould].Cmd.arrbModuloPoint[i2]:=FALSE;	
	END_IF		
END_FOR
//////////////裁切////////////
FOR i2:=0 TO 10 BY 1 DO			
	IF arrAxisCtrl[AxisNo.Cuter].Cmd.arrbModuloGo[i2] AND arrAxis[AxisNo.Cuter].Status.StandStill THEN		
		IF NOT arrAxisCtrl[AxisNo.Cuter].Cmd.arrbModuloPoint[i2] THEN	
			arrAxisCtrl[AxisNo.Cuter].Cmd.fPositon_of_Mod:=arrAxisPar[AxisNo.Cuter].arrTargetPoint[i2];//绝对模长位置定位
			arrAxisCtrl[AxisNo.Cuter].Cmd.bMoveModulo:=TRUE;
			arrAxisCtrl[AxisNo.Cuter].Cmd.arrbModuloGo[i2]:=FALSE;
		ELSE	
			arrAxisCtrl[AxisNo.Cuter].Cmd.arrbModuloGo[i2]:=FALSE;
		END_IF	
	END_IF		
	IF arrAxisPar[AxisNo.Cuter].arrTargetPoint[i2]-0.1<= arrAxisCtrl[AxisNo.Cuter].Status.fModuloActPos AND		
		arrAxisPar[AxisNo.Cuter].arrTargetPoint[i2]+0.1>=arrAxisCtrl[AxisNo.Cuter].Status.fModuloActPos AND	
		NOT arrAxisCtrl[AxisNo.Cuter].Cmd.bMoveModulo THEN	
		arrAxisCtrl[AxisNo.Cuter].Cmd.arrbModuloPoint[i2]:=TRUE;	
	ELSE		
		arrAxisCtrl[AxisNo.Cuter].Cmd.arrbModuloPoint[i2]:=FALSE;	
	END_IF		
END_FOR			
//////////////CCD压片升降////////////
FOR i2:=0 TO 10 BY 1 DO			
	IF arrAxisCtrl[AxisNo.CCDPressPush].Cmd.arrbModuloGo[i2] AND arrAxis[AxisNo.CCDPressPush].Status.StandStill THEN		
		IF NOT arrAxisCtrl[AxisNo.CCDPressPush].Cmd.arrbModuloPoint[i2] THEN	
			arrAxisCtrl[AxisNo.CCDPressPush].Cmd.fPositon_of_Mod:=arrAxisPar[AxisNo.CCDPressPush].arrTargetPoint[i2];//绝对模长位置定位
			arrAxisCtrl[AxisNo.CCDPressPush].Cmd.bMoveModulo:=TRUE;
			arrAxisCtrl[AxisNo.CCDPressPush].Cmd.arrbModuloGo[i2]:=FALSE;
		ELSE	
			arrAxisCtrl[AxisNo.CCDPressPush].Cmd.arrbModuloGo[i2]:=FALSE;
		END_IF	
	END_IF		
	IF arrAxisPar[AxisNo.CCDPressPush].arrTargetPoint[i2]-0.1<= arrAxisCtrl[AxisNo.CCDPressPush].Status.fModuloActPos AND		
		arrAxisPar[AxisNo.CCDPressPush].arrTargetPoint[i2]+0.1>=arrAxisCtrl[AxisNo.CCDPressPush].Status.fModuloActPos AND	
		NOT arrAxisCtrl[AxisNo.CCDPressPush].Cmd.bMoveModulo THEN	
		arrAxisCtrl[AxisNo.CCDPressPush].Cmd.arrbModuloPoint[i2]:=TRUE;	
	ELSE		
		arrAxisCtrl[AxisNo.CCDPressPush].Cmd.arrbModuloPoint[i2]:=FALSE;	
	END_IF		
END_FOR						


///////////////////////////////////////////////////////////纠偏控制信号自动复位///////////////////////////////////////////////////////////////////
IF tonCondition[5].Q THEN
	arrRecCtrl[RecNo.PoleWind].Cmd.bCentre:=FALSE;
END_IF
IF tonCondition[6].Q THEN
	arrRecCtrl[RecNo.PoleWind].Cmd.bAuto:=FALSE;
END_IF
IF tonCondition[7].Q THEN
	arrRecCtrl[RecNo.PoleWind].Cmd.bManual:=FALSE;
END_IF
IF tonCondition[8].Q THEN
	arrRecCtrl[RecNo.PoleProcess].Cmd.bCentre:=FALSE;
END_IF
IF tonCondition[9].Q THEN
	arrRecCtrl[RecNo.PoleProcess].Cmd.bAuto:=FALSE;
END_IF
IF tonCondition[10].Q THEN
	arrRecCtrl[RecNo.PoleProcess].Cmd.bManual:=FALSE;
END_IF

///////////////////////////////////////////////////////////切刀计数///////////////////////////////////////////////////////////////////
rtCount1(CLK:=arrAxisCtrl[AxisNo.Mould].Status.fModuloActPos>=170 AND arrAxisCtrl[AxisNo.Mould].Status.fModuloActPos<=190);
IF rtCount1.Q THEN
	PolePar.iMouldCount1:=PolePar.iMouldCount1+1;
	PolePar.iMouldCount2:=PolePar.iMouldCount2+1;
	IF iPartSelect =1 THEN
			YL_GVL2[1]:=YL_GVL2[1]+1;
	ELSIF iPartSelect =2 THEN
			YL_GVL2[3]:=YL_GVL2[3]+1;
	END_IF

END_IF

IF rtCount2.Q THEN
	PolePar.iCuterCount:=PolePar.iCuterCount+1;
END_IF
///////////////////////////////////////////////////////////切刀计数清零//////////////////////////////////////////////////////////
rtMouldClear1( CLK := PolePar.iMouldclear1    ); //前模具切刀
rtMouldClear2( CLK := PolePar.iMouldclear2    );  //后模具切刀   
rtCuterClear( CLK := PolePar.iCuterclear    );    
IF rtMouldClear1.Q THEN          //前倒角模具切刀清零
	PolePar.iMouldCount1:=0;
END_IF
IF rtMouldClear2.Q THEN          //后倒角模具切刀清零
	PolePar.iMouldCount2:=0;
END_IF
IF rtCuterClear.Q THEN          //裁切切刀清零
	PolePar.iCuterCount:=0;
END_IF




